(* Logix 5000 project; controller L3 vendor 1 type 14 code 92 rev 20.12; software revision 20.04 *)

TASK _11_PID2 (periodic, rate 100 ms, priority 14, watchdog 500 ms) : _11_PID2
TASK main (periodic, rate 100 ms, priority 13, watchdog 500 ms) : _2_GENERAL
TASK MainTask (continuous, watchdog 500 ms) : MainProgram
TASK pid_lent (periodic, rate 1000 ms, priority 15, watchdog 500 ms) : pid_dec

MODULES
   Local : vendor 1 type 14 code 92 (ICP 0, rev 20.12)
       : 1756-IB16 (ICP 1, rev 3.1, Input RPI 20 ms)
           Local:1:I.DATA.8   // pmp run
       : 1756-OB32 (ICP 3, rev 3.1, Output RPI 20 ms)
           Local:3:O.DATA.0   // START/STOP DRIVE POMP WKK
           Local:3:O.DATA.1   // VRIJGAVE POMP WKK
       : 1756-IF8 (ICP 2, rev 1.1, Input RPI 200 ms)
       : 1756-OF4 (ICP 4, rev 1.1, Output RPI 100 ms)
      L3_usine : 1756-EN2T (ICP 6, Ethernet 192.168.3.161, rev 2.1)
         STAT_usine : 1756-ENBT (Ethernet 192.168.3.162, rev 6.1)
            STAT : 1756-L72 (ICP 0, rev 20.1, $879c264d$ RPI 250 ms)
         EtherNet_Bridge : 1756-ENBT (Ethernet 192.168.3.150, rev 4.3, Output RPI 10 ms)
            WKK : vendor 1 type 14 code 92 (ICP 2, rev 20.12, $f706532b$ RPI 250 ms)
      IO : 1756-EN2T (ICP 5, Ethernet 192.168.1.2, rev 2.1)
         IO_decap : 1794-AENTR (Ethernet 192.168.1.6, rev 1.1, Output RPI 20 ms)
            decap_DO_3 : vendor 1 type 7 code 35 (Flex 3, rev 1.1)
            decap_DI_2 : 1794-IB16 (Flex 2, rev 1.1)
            decap_AI_0 : vendor 1 type 10 code 30 (Flex 0, rev 1.1, Input RPI 80 ms)
            decap_AO_1 : vendor 1 type 10 code 31 (Flex 1, rev 1.1, Output RPI 80 ms)
         R2 : vendor 1 type 12 code 228 (Ethernet 192.168.1.4, rev 1.1)
             : vendor 1 type 117 code 6 (SLCChassis 10, rev 1.1, StandardDataDriven RPI 20 ms)
             : vendor 1 type 117 code 6 (SLCChassis 9, rev 1.1, StandardDataDriven RPI 20 ms)
             : vendor 1 type 116 code 24 (SLCChassis 2, rev 1.1, StandardDataDriven RPI 20 ms)
                 R2:2:O.DATA.0   // CONSIGNE SORTIE -5% pg78
                 R2:2:O.DATA.1   // CONSIGNE SORTIE +5% pg78
                 R2:2:O.DATA.2   // CONSIGNE SORTIE -20% pg78
                 R2:2:O.DATA.3   // CONSIGNE SORTIE +20% pg78
                 R2:2:O.DATA.4   // CONSIGNE SORTIE 0 pg78
                 R2:2:O.DATA.5   // LP8 POTENTIOMETRE ENR POSITION incorrecte pg80
                 R2:2:O.DATA.6   // POTENTIOMETRE ENROULEUSE MIN pg80
                 R2:2:O.DATA.7   // LP6 TRS ACCU EXTREME VIDE pg82
                 R2:2:O.DATA.8   // TRS pg83
                 R2:2:O.DATA.9   // JOG -> BS4 pg85
                 R2:2:O.DATA.10   // JOG <- BS4 pg85
                 R2:2:O.DATA.11   // VERROUILAGE CISAILLE SORTIE pg87
                 R2:2:O.DATA.12   // REGLAGE TRACTION pg 93
                 R2:2:O.DATA.13   // QUEUE DE BANDE ENROULEUSE pg94
                 R2:2:O.DATA.14   // JOG -> ENR pg94.1
                 R2:2:O.DATA.15   // JOG <- ENR pg94.1
                 R2:2:O.POINT_0   // n,bvch
             : vendor 1 type 116 code 24 (SLCChassis 6, rev 1.1, StandardDataDriven RPI 20 ms)
                 R2:6:O.DATA.0   // lampe verte
                 R2:6:O.DATA.1   // bell
                 R2:6:O.DATA.2   // lampe orange
                 R2:6:O.DATA.3   // lampe rouge
                 R2:6:O.DATA.4   // lampe bleu
                 R2:6:O.DATA.5   // vann apport soude décapage
                 R2:6:O.DATA.6   // res
                 R2:6:O.DATA.7   // res
                 R2:6:O.DATA.8   // res
                 R2:6:O.DATA.9   // res
                 R2:6:O.DATA.10   // res
                 R2:6:O.DATA.11   // res
                 R2:6:O.DATA.12   // res
                 R2:6:O.DATA.13   // res
                 R2:6:O.DATA.14   // res
                 R2:6:O.DATA.15   // reserve pour vanne acide
                 R2:6:O.POINT_0   // lampe verte
                 R2:6:O.POINT_1   // bell
                 R2:6:O.POINT_2   // lampe orange
                 R2:6:O.POINT_3   // lampe rouge
                 R2:6:O.POINT_4   // lampe bleu
                 R2:6:O.POINT_5   // vann apport soude décapage
                 R2:6:O.POINT_15   // reserve pour vanne acide
             : vendor 1 type 116 code 3 (SLCChassis 7, rev 1.1, StandardDataDriven RPI 20 ms)
                 R2:7:I.DATA.0   // vanne apport soude ouverte
                 R2:7:I.DATA.1   // vanne apport soude fermée
                 R2:7:I.DATA.2   // t° redresseur T1 R2
                 R2:7:I.DATA.3   // t° redresseur T2 R2
                 R2:7:I.DATA.4   // t° redresseur T1 R3
                 R2:7:I.DATA.5   // t° redresseur T2 R3
                 R2:7:I.DATA.6   // t° redresseur T1 R4
                 R2:7:I.DATA.7   // t° redresseur T2 R4
                 R2:7:I.DATA.8   // t° redresseur T1 R1
                 R2:7:I.DATA.9   // t° redresseur T2 R1
                 R2:7:I.POINT_0   // vanne apport soude ouverte
                 R2:7:I.POINT_1   // vanne apport soude fermée
                 R2:7:I.POINT_2   // t° redresseur T1 R2
                 R2:7:I.POINT_3   // t° redresseur T2 R2
                 R2:7:I.POINT_4   // t° redresseur T1 R3
                 R2:7:I.POINT_5   // t° redresseur T2 R3
                 R2:7:I.POINT_6   // t° redresseur T1 R4
                 R2:7:I.POINT_7   // t° redresseur T2 R4
                 R2:7:I.POINT_8   // t° redresseur T1 R1
                 R2:7:I.POINT_9   // t° redresseur T2 R1
             : vendor 1 type 116 code 3 (SLCChassis 1, rev 1.1, StandardDataDriven RPI 20 ms)
                 R2:1:I.DATA.0   // TRE ACCU EXTREMEVIDE
                 R2:1:I.DATA.1   // TRE en SERVICE
                 R2:1:I.DATA.2   // TRE MAN/COORD.
                 R2:1:I.DATA.3   // AUTORISATION JOG BS2
                 R2:1:I.DATA.4   // AUTORISATION JOG BS3
                 R2:1:I.DATA.5   // MARCHE SORTIE
                 R2:1:I.DATA.6   // MARCHE SORTIE
                 R2:1:I.DATA.7   // ARRET SORTIE
                 R2:1:I.DATA.8   // SORTIE COORD.
                 R2:1:I.DATA.9   // SORTIE MANU
                 R2:1:I.DATA.10   // REPRISE MANU SORTIE
                 R2:1:I.DATA.11   // ENR POTENT.POSITION MAX
                 R2:1:I.DATA.12   // ENR POTENT.POSITION MIN
                 R2:1:I.DATA.13   // TRS RALENTSSEMENT
                 R2:1:I.DATA.14   // TRS POSITION TRAVAIL ARRIERE
                 R2:1:I.DATA.15   // TRS POSITION TRAVAIL AVANT
                 R2:1:I.POINT_0   // tdwsrdrw
             : vendor 1 type 117 code 6 (SLCChassis 8, rev 1.1, StandardDataDriven RPI 20 ms)
             : vendor 1 type 116 code 3 (SLCChassis 3, rev 1.1, StandardDataDriven RPI 20 ms)
                 R2:3:I.DATA.0   // TRS ACCU VIDE
                 R2:3:I.DATA.1   // TRS ACCU REMPLI
                 R2:3:I.DATA.2   // TRS ACCU REMPLI EXTREME
                 R2:3:I.DATA.3   // TRS ACCU VIDE EXTREME
                 R2:3:I.DATA.4   // TRS en service
                 R2:3:I.DATA.5   // TRS
                 R2:3:I.DATA.6   // JOG -> BS4
                 R2:3:I.DATA.7   // JOG <- BS4
                 R2:3:I.DATA.8   // BS4M N=0
                 R2:3:I.DATA.9   // BS3M N=0
                 R2:3:I.DATA.10   // QUEUE DE BANDE ENROULEUSE ON
                 R2:3:I.DATA.11   // QUEUE DE BANDE ENROULEUSE OFF
                 R2:3:I.DATA.12   // JOG -> ENR
                 R2:3:I.DATA.13   // JOG <- ENR
                 R2:3:I.DATA.14   // BP POSITIONNER ENR
                 R2:3:I.DATA.15   // ENROULEUSE POSITIONNEE
             : vendor 1 type 117 code 11 (SLCChassis 11, rev 1.1, StandardDataDriven RPI 20 ms)
             : vendor 1 type 116 code 3 (SLCChassis 5, rev 1.1, StandardDataDriven RPI 20 ms)
                 R2:5:I.DATA.0   // N=0 ENR
                 R2:5:I.DATA.1   // RAZ DIAMETRE ENROULEUSE
                 R2:5:I.DATA.2   // MANDRIN EXPANSE
                 R2:5:I.DATA.3   // ready drive ventilateur 03
                 R2:5:I.DATA.4   // ready drive ventilateur 2
                 R2:5:I.DATA.5   // ready drive ventilateur 01
                 R2:5:I.DATA.6   // protection drive ventilateur 03
                 R2:5:I.DATA.7   // protection drive ventilateur 2
                 R2:5:I.DATA.8   // protection drive ventilateur 01
                 R2:5:I.POINT_0   // N=0 ENR
                 R2:5:I.POINT_1   // RAZ DIAMETRE ENROULEUSE
                 R2:5:I.POINT_2   // MANDRIN EXPANSE
                 R2:5:I.POINT_3   // ready drive ventilateur 03
                 R2:5:I.POINT_4   // ready drive ventilateur 2
                 R2:5:I.POINT_5   // ready drive ventilateur 01
                 R2:5:I.POINT_6   // protection drive ventilateur 03
                 R2:5:I.POINT_7   // protection drive ventilateur 2
                 R2:5:I.POINT_8   // protection drive ventilateur 01
             : vendor 1 type 116 code 24 (SLCChassis 4, rev 1.1, StandardDataDriven RPI 20 ms)
                 R2:4:O.DATA.0   // POSITIONNER MANDRIN ENR pg94.1
                 R2:4:O.DATA.1   // RAZ DIAMETRE ENR pg96
                 R2:4:O.DATA.2   // klaxon demarrage ligne
                 R2:4:O.DATA.3   // M/A VENTILATEUR 03
                 R2:4:O.DATA.4   // M/A VENTILATEUR 2
                 R2:4:O.DATA.5   // M/A VENTILATEUR 01
                 R2:4:O.DATA.6   // VANNE VIDANGE TOURS
                 R2:4:O.DATA.7   // M/A PMP DOSEUSE TOUR REFROIDISSEMENT
                 R2:4:O.POINT_0   // POSITIONNER MANDRIN ENR pg94.1
                 R2:4:O.POINT_1   // RAZ DIAMETRE ENR pg96
                 R2:4:O.POINT_2   // klaxon demarrage ligne
                 R2:4:O.POINT_3   // M/A VENTILATEUR 03
                 R2:4:O.POINT_4   // M/A VENTILATEUR 2
                 R2:4:O.POINT_5   // M/A VENTILATEUR 01
                 R2:4:O.POINT_6   // VANNE VIDANGE TOURS
                 R2:4:O.POINT_7   // M/A PMP DOSEUSE TOUR REFROIDISSEMENT
         R1 : vendor 1 type 12 code 228 (Ethernet 192.168.1.3, rev 1.1)
             : vendor 1 type 116 code 3 (SLCChassis 6, rev 1.1, StandardDataDriven RPI 20 ms)
                 R1:6:I.DATA.0   // DEFAUT CONVERTISSEUR
                 R1:6:I.DATA.1   // ACQUIT KLAXON
                 R1:6:I.DATA.2   // TENSION 24 V PAS OK
                 R1:6:I.DATA.3   // N>N0
                 R1:6:I.DATA.4   // RUPTURE BANDE ENTREE
                 R1:6:I.DATA.5   // RUPTURE BANDE SORTIE
                 R1:6:I.DATA.6   // FREIN DEROULEUSE 1
                 R1:6:I.DATA.7   // FREIN DEROULEUSE 2
                 R1:6:I.DATA.8   // JOG <- BS1 + DEC
                 R1:6:I.DATA.9   // JOG -> BS1 + DEC
                 R1:6:I.DATA.10   // JOG <- DEC
                 R1:6:I.DATA.11   // JOG -> DEC
                 R1:6:I.DATA.12   // DEC N<N0
                 R1:6:I.DATA.13   // BS1M N<N0
                 R1:6:I.DATA.14   // BS2M N<N0
                 R1:6:I.DATA.15   // CISAILLE ENTREE BASSE
                 R1:6:I.POINT_0   // dsgt erqe
             : vendor 1 type 116 code 24 (SLCChassis 7, rev 1.1, StandardDataDriven RPI 20 ms)
                 R1:7:O.DATA.0   // RUN TEMPO pg38
                 R1:7:O.DATA.1   // FERMER PINCEUR pg39
                 R1:7:O.DATA.2   // LP6 RUPTURE BANDE pg39
                 R1:7:O.DATA.3   // JOG -> DEC pg55
                 R1:7:O.DATA.4   // JOG <- DEC pg55
                 R1:7:O.DATA.5   // N<N0 DEC pg57
                 R1:7:O.DATA.6   // LP4 M/A ENTREE pg60
                 R1:7:O.DATA.7   // LP4 ENTREE COORDONNEE pg61
                 R1:7:O.DATA.8   // LP4 ENTREE MANUEL pg61
                 R1:7:O.DATA.9   // MAN/COORD. ENTREE pg62
                 R1:7:O.DATA.10   // CONSIGNE ENTREE-5% pg63
                 R1:7:O.DATA.11   // CONSIGNE ENTREE+5% pg63
                 R1:7:O.DATA.12   // CONSIGNE ENTREE-20% pg63
                 R1:7:O.DATA.13   // CONSIGNE ENTREE+20% pg63
                 R1:7:O.DATA.14   // CONSIGNE ENTREE pg63
                 R1:7:O.DATA.15   // JOG <- BS1 pg66
                 R1:7:O.POINT_0   // vgcf
             : vendor 1 type 116 code 3 (SLCChassis 3, rev 1.1, StandardDataDriven RPI 20 ms)
                 R1:3:I.DATA_0   // EMG 2
                 R1:3:I.DATA_1   // EMG 3
                 R1:3:I.DATA_10   // TRE PRET REFERENCE
                 R1:3:I.DATA_11   // BS2M PRET REFERENCE
                 R1:3:I.DATA_12   // BS3M PRET REFERENCE
                 R1:3:I.DATA_13   // TRS PRET REFERENCE
                 R1:3:I.DATA_14   // BS4M PRET REFERENCE
                 R1:3:I.DATA_15   // ENR PRET REFERENCE
                 R1:3:I.DATA_2   // bp marche ligne
                 R1:3:I.DATA_3   // BP STOP
                 R1:3:I.DATA_4   // DEC ENCLENCHE
                 R1:3:I.DATA_5   // LIGNE ENCLENCHEE
                 R1:3:I.DATA_6   // READY FOR RUN
                 R1:3:I.DATA_7   // BP RUN
                 R1:3:I.DATA_8   // AEC PRET REFERENCE
                 R1:3:I.DATA_9   // BS1M PRET REFERENCE
                 R1:3:I.POINT_0   // dxfh
             : vendor 1 type 116 code 3 (SLCChassis 1, rev 1.1, StandardDataDriven RPI 20 ms)
                 R1:1:I.DATA.0   // bp start groupe hydraulique entrée
                 R1:1:I.DATA.1   // bp stop groupe hydraulique entrée
                 R1:1:I.DATA.2   // pression groupe hydraulique entrée 100 bars
                 R1:1:I.DATA.3   // pression groupe hydraulique entrée 70 bars
                 R1:1:I.DATA.4   // niveau groupe hydraulique entrée
                 R1:1:I.DATA.5   // by pass groupe hydraulique entrée
                 R1:1:I.DATA.6   // by pass groupe hydraulique sortie
                 R1:1:I.DATA.7   // bp start groupe hydraulique sortie
                 R1:1:I.DATA.8   // bp stop groupe hydraulique sortie
                 R1:1:I.DATA.9   // 100 BARS GROUPE HYDR.SORTIE
                 R1:1:I.DATA.10   // pression groupe hydraulique sortie 70 bars
                 R1:1:I.DATA.11   // niveau groupe hydraulique sortie
                 R1:1:I.DATA.12   // réarmement signalisation
                 R1:1:I.DATA.13   // pressostat air comprimé
                 R1:1:I.DATA.14   // centrage ok
                 R1:1:I.DATA.15   // centrage EMG 1
                 R1:1:I.POINT_0   // bp start groupe hydraulique entrée
                 R1:1:I.POINT_1   // bp stop groupe hydraulique entrée
                 R1:1:I.POINT_2   // pression groupe hydraulique entrée 100 bars
                 R1:1:I.POINT_3   // pression groupe hydraulique entrée 70 bars
                 R1:1:I.POINT_4   // niveau groupe hydraulique entrée
                 R1:1:I.POINT_6   // by pass groupe hydraulique sortie
                 R1:1:I.POINT_5   // by pass groupe hydraulique entrée
                 R1:1:I.POINT_7   // bp start groupe hydraulique sortie
                 R1:1:I.POINT_8   // bp stop groupe hydraulique sortie
                 R1:1:I.POINT_9   // 100 BARS GROUPE HYDR.SORTIE
                 R1:1:I.POINT_10   // pression groupe hydraulique sortie 70 bars
                 R1:1:I.POINT_11   // niveau groupe hydraulique sortie
                 R1:1:I.POINT_12   // réarmement signalisation
                 R1:1:I.POINT_13   // pressostat air comprimé
                 R1:1:I.POINT_14   // centrage ok
                 R1:1:I.POINT_15   // centrage EMG 1
             : vendor 1 type 116 code 24 (SLCChassis 9, rev 1.1, StandardDataDriven RPI 20 ms)
                 R1:9:O.DATA.0   // JOG -> BS1 pg66
                 R1:9:O.DATA.1   // LP4 TRE RALENTISSEMENT pg68
                 R1:9:O.DATA.2   // LP6 TRE ACCU VIDE pg69
                 R1:9:O.DATA.3   // TRE MAN/COORDON. pg70
                 R1:9:O.DATA.4   // AUTORISATION JOG BS2 pg 72
                 R1:9:O.DATA.5   // AUTORISATION JOG BS3 pg70
                 R1:9:O.DATA.6   // LP8 MARCHE SORTIE pg74
                 R1:9:O.DATA.7   // LP7 MARCHE SORTIE pg74
                 R1:9:O.DATA.8   // LP7 SORTIE MANU pg75
                 R1:9:O.DATA.9   // LP7 SORTIE COORD. pg75
                 R1:9:O.DATA.10   // LP8 NOUVELLE BOBINE SORTIE pg75
                 R1:9:O.DATA.11   // ENR DEBUT FIN DE BOBINE pg76
                 R1:9:O.DATA.12   // CONS. SORTIE MAN/COORD. pg77
                 R1:9:O.DATA.13   // CONSIGNE SORTIE MANU pg77
                 R1:9:O.DATA.14   // CONSIGNE SORTIE MARCHE MANU pg77
                 R1:9:O.DATA.15   // CONSIGNE SORTIE pg77
                 R1:9:O.POINT_0   // hfgfh
             : vendor 1 type 116 code 24 (SLCChassis 4, rev 1.1, StandardDataDriven RPI 20 ms)
                 R1:4:O.DATA.0   // DRIVE ON pg16.1
                 R1:4:O.DATA.1   // ARRET pg17
                 R1:4:O.DATA.2   // AUXILIAIRE 1 ARRET pg17
                 R1:4:O.DATA.3   // AUXILIAIRE 2 ARRET pg17
                 R1:4:O.DATA.4   // LP6 DRIVE ENCLENCHE pg18
                 R1:4:O.DATA.5   // LP6 READY FOR RUN pg18.1
                 R1:4:O.DATA.6   // RUN pg20
                 R1:4:O.DATA.7   // MARCHE SYNCHRO DEC pg21
                 R1:4:O.DATA.8   // MARCHE SYNCHRO BS1 pg21
                 R1:4:O.DATA.9   // MARCHE SYNCHRO TRE pg21
                 R1:4:O.DATA.10   // MARCHE SYNCHRO BS2 pg21
                 R1:4:O.DATA.11   // MARCHE SYNCHRO BS3 pg21
                 R1:4:O.DATA.12   // MARCHE SYNCHRO TRS pg21
                 R1:4:O.DATA.13   // MARCHE SYNCHRO BS4 pg21
                 R1:4:O.DATA.14   // MARCHE SYNCHRO ENR pg21
                 R1:4:O.DATA.15   // LP6 MARCHE COORDONNEE pg22
                 R1:4:O.POINT_0   // n cb
             : vendor 1 type 116 code 3 (SLCChassis 8, rev 1.1, StandardDataDriven RPI 20 ms)
                 R1:8:I.DATA.0   // TABLE CISAILLE ENTREE OK
                 R1:8:I.DATA.1   // BP MARCHE ENTREE
                 R1:8:I.DATA.2   // BP MARCHE ENTREE
                 R1:8:I.DATA.3   // BP ARRET ENTREE
                 R1:8:I.DATA.4   // BP ENTREE COORDONNE
                 R1:8:I.DATA.5   // BP ENTREE MANU
                 R1:8:I.DATA.6   // POTENTIOMETRE ENTREE POSITION MAX
                 R1:8:I.DATA.7   // POTENTIOMETRE ENTREE POSITION MIN
                 R1:8:I.DATA.8   // JOG <-BS1
                 R1:8:I.DATA.9   // JOG ->BS1
                 R1:8:I.DATA.10   // TRE RALENTISSEMENT
                 R1:8:I.DATA.11   // TRE POSITION TRAVAIL AVANT
                 R1:8:I.DATA.12   // TRE POSITION TRAVAIL ARRIERE
                 R1:8:I.DATA.13   // TRE ACCU REMPLI
                 R1:8:I.DATA.14   // TRE ACCU VIDE
                 R1:8:I.DATA.15   // TRE ACCU EXTREME REMPLI
                 R1:8:I.POINT_0   // ;,vn
            O2 : vendor 1 type 116 code 24 (SLCChassis 2, rev 1.1, StandardDataDriven RPI 20 ms)
                 R1:2:O.DATA.0   // n<n0 pg37
                 R1:2:O.DATA.1   // LP6 marche groupe hydraulique entrée pg8
                 R1:2:O.DATA.2   // marche groupe hydraulique entrée pg11
                 R1:2:O.DATA.3   // autorisation alimentation tension de groupe Hydraulique entrée
                 R1:2:O.DATA.4   // vanne mise en pression groupe hydraumique entrée pg8
                 R1:2:O.DATA.5   // LP6 marche groupe hydraulique sortie pg9
                 R1:2:O.DATA.6   // marche groupe hydraulique sortie pg11
                 R1:2:O.DATA.7   // autorisation alimentation tension de groupe Hydraulique sortie
                 R1:2:O.DATA.8   // vanne mise en pression groupe hydraumique sortie pg9
                 R1:2:O.DATA.9   // LP6 defaut pression groupe hydraulique entrée pg10
                 R1:2:O.DATA.10   // LP6 défaut niveau groupe hydraulique entrée pg10
                 R1:2:O.DATA.11   // LP6 défaut pression groupe hydraulique sortie 70 bars
                 R1:2:O.DATA.12   // LP6 défaut niveau groupe hydraulique entrée pg10
                 R1:2:O.DATA.13   // LP6 défaut pression air comprimé pg11.1
                 R1:2:O.DATA.14   // drive on pg16
                 R1:2:O.DATA.15   // LP6 demande drive on
                 R1:2:O.POINT_0   // n<n0 pg37
                 R1:2:O.POINT_1   // LP6 marche groupe hydraulique entrée pg8
                 R1:2:O.POINT_2   // marche groupe hydraulique entrée pg11
                 R1:2:O.POINT_3   // autorisation alimentation tension de groupe Hydraulique entrée
                 R1:2:O.POINT_4   // vanne mise en pression groupe hydraumique entrée pg8
                 R1:2:O.POINT_5   // LP6 marche groupe hydraulique sortie pg9
                 R1:2:O.POINT_6   // marche groupe hydraulique sortie pg11
                 R1:2:O.POINT_7   // autorisation alimentation tension de groupe Hydraulique sortie
                 R1:2:O.POINT_8   // vanne mise en pression groupe hydraumique sortie pg9
                 R1:2:O.POINT_9   // LP6 defaut pression groupe hydraulique entrée pg10
                 R1:2:O.POINT_10   // LP6 défaut niveau groupe hydraulique entrée pg10
                 R1:2:O.POINT_12   // LP6 défaut niveau groupe hydraulique entrée pg10
                 R1:2:O.POINT_11   // LP6 défaut pression groupe hydraulique sortie 70 bars
                 R1:2:O.POINT_14   // drive on pg16
                 R1:2:O.POINT_13   // LP6 défaut pression air comprimé pg11.1
                 R1:2:O.POINT_15   // LP6 demande drive on
             : vendor 1 type 116 code 24 (SLCChassis 5, rev 1.1, StandardDataDriven RPI 20 ms)
                 R1:5:O.DATA.0   // LP6 PRET REFERENCE DEC pg25
                 R1:5:O.DATA.1   // LP6 PRET REFERENCE BS1 pg25
                 R1:5:O.DATA.2   // LP6 PRET REFERENCE TRE pg25
                 R1:5:O.DATA.3   // LP6 PRET REFERENCE BS2 pg25
                 R1:5:O.DATA.4   // LP6 PRET REFERENCE BS3 pg25
                 R1:5:O.DATA.5   // LP6 PRET REFERENCE TRS pg25
                 R1:5:O.DATA.6   // LP6 PRET REFERENCE BS4 pg25
                 R1:5:O.DATA.7   // LP6 PRET REFERENCE ENR pg25
                 R1:5:O.DATA.8   // LP6 PRET REFERENCE LIGNE pg25
                 R1:5:O.DATA.9   // LIGNE PRET REFERENCE pg26
                 R1:5:O.DATA.10   // LP6 DEFAUT PRET REFERENCE pg27
                 R1:5:O.DATA.11   // LP6 DEFAUT PRET REFERENCE BS2 BS3 pg27
                 R1:5:O.DATA.12   // LP6 DEFAUT MISE EN VITESSE pg27
                 R1:5:O.DATA.13   // LP6 DEFAUT CONVERTISSEUR pg28
                 R1:5:O.DATA.14   // KLAXON pg30
                 R1:5:O.DATA.15   // LP6 ALIM. 24 V OK pg33
                 R1:5:O.POINT_0   // ;: ,hwfd
         R3 : vendor 1 type 12 code 228 (Ethernet 192.168.1.5, rev 1.1)
             : vendor 1 type 116 code 6 (SLCChassis 7, rev 1.1, StandardDataDriven RPI 20 ms)
                 R3:7:I.POINT_0   // v cxbvwc
             : vendor 1 type 117 code 11 (SLCChassis 2, rev 1.1, StandardDataDriven RPI 20 ms)
                 R3:2:O.CHANNEL_0_OUTPUT   // wxvc<
             : vendor 1 type 117 code 6 (SLCChassis 6, rev 1.1, StandardDataDriven RPI 20 ms)
                 R3:6:I.CHANNEL_0_DATA   // vwx
             : vendor 1 type 117 code 6 (SLCChassis 3, rev 1.1, StandardDataDriven RPI 20 ms)
                 R3:3:I.CHANNEL_0_DATA   // vwxc
             : vendor 1 type 116 code 6 (SLCChassis 4, rev 1.1, StandardDataDriven RPI 20 ms)
                 R3:4:I.DATA.0   // vanne chauffe degrai open
                 R3:4:I.DATA.1   // vanne chauffe degrai closed
                 R3:4:I.DATA.2   // vanne chauffe decapa open
                 R3:4:I.DATA.3   // vanne chauffe decapa close
                 R3:4:I.DATA.4   // vanne froid decapage open
                 R3:4:I.DATA.5   // vanne froid decapage closed
                 R3:4:I.DATA.6   // fc open vanne ano
                 R3:4:I.DATA.7   // fc closed vanne ano
                 R3:4:I.DATA.8   // vanne chauffage colm open
                 R3:4:I.DATA.9   // vanne chauffage colm closed
                 R3:4:I.DATA.10   // vanne 2 chauffage co open
                 R3:4:I.DATA.11   // vanne 2 chauffage co closed
                 R3:4:I.DATA.12   // P1 T37 DECAPAGE RUN
                 R3:4:I.DATA.13   // P1 T37 DECAPAGE PROTECTION
                 R3:4:I.DATA.14   // P2 DECAPAGE RUN
                 R3:4:I.DATA.15   // P2 DECAPAGE PROTECTION
                 R3:4:I.DATA.16   // Naoh L3VA1 FC O
                 R3:4:I.DATA.17   // Naoh L3VA1 FC f
                 R3:4:I.DATA.18   // Naoh L3VA2 FC O
                 R3:4:I.DATA.19   // Naoh L3VA2 FC F
                 R3:4:I.DATA.20   // Naoh L3VA3 FC O
                 R3:4:I.DATA.21   // Naoh L3VA3 FC F
                 R3:4:I.DATA.22   // Naoh L3VA4 FC O
                 R3:4:I.DATA.23   // Naoh L3VA4 FC F
                 R3:4:I.DATA.24   // re
                 R3:4:I.DATA.25   // re
                 R3:4:I.DATA.26   // NaOH FLOW METER PULSE 0.1 M³
                 R3:4:I.DATA.27   // laveur fumée ok
                 R3:4:I.DATA.28   // fc vanne apport acide ano open
                 R3:4:I.DATA.29   // fc vanne apport acide ano close
                 R3:4:I.DATA.30   // fc vanne apport acide neutral open
                 R3:4:I.DATA.31   // fc vanne apport acide neutral close
                 R3:4:I.POINT_0   // vanne chauffe degrai open
                 R3:4:I.POINT_1   // vanne chauffe degrai closed
                 R3:4:I.POINT_2   // vanne chauffe decapa open
                 R3:4:I.POINT_3   // vanne chauffe decapa close
                 R3:4:I.POINT_4   // vanne froid decapage open
                 R3:4:I.POINT_5   // vanne froid decapage closed
                 R3:4:I.POINT_6   // fc open vanne ano
                 R3:4:I.POINT_7   // fc closed vanne ano
                 R3:4:I.POINT_8   // vanne chauffage colm open
                 R3:4:I.POINT_9   // vanne chauffage colm closed
                 R3:4:I.POINT_10   // vanne 2 chauffage co open
                 R3:4:I.POINT_11   // vanne 2 chauffage co closed
                 R3:4:I.POINT_12   // P1 T37 DECAPAGE RUN
                 R3:4:I.POINT_13   // P1 T37 DECAPAGE PROTECTION
                 R3:4:I.POINT_14   // P2 DECAPAGE RUN
                 R3:4:I.POINT_15   // P2 DECAPAGE PROTECTION
                 R3:4:I.POINT_16   // Naoh L3VA1 FC O
                 R3:4:I.POINT_17   // Naoh L3VA1 FC f
                 R3:4:I.POINT_18   // Naoh L3VA2 FC O
                 R3:4:I.POINT_19   // Naoh L3VA2 FC F
                 R3:4:I.POINT_20   // Naoh L3VA3 FC O
                 R3:4:I.POINT_21   // Naoh L3VA3 FC F
                 R3:4:I.POINT_22   // Naoh L3VA4 FC O
                 R3:4:I.POINT_23   // Naoh L3VA4 FC F
                 R3:4:I.POINT_26   // NaOH FLOW METER PULSE 0.1 M³
                 R3:4:I.POINT_27   // laveur fumée ok
                 R3:4:I.POINT_24   // fc vanne apport acide ano open
                 R3:4:I.POINT_28   // fc vanne apport acide ano open
                 R3:4:I.POINT_29   // fc vanne apport acide ano close
                 R3:4:I.POINT_30   // fc vanne apport acide neutral open
                 R3:4:I.POINT_31   // fc vanne apport acide neutral close
             : vendor 1 type 117 code 11 (SLCChassis 1, rev 1.1, StandardDataDriven RPI 20 ms)
                 R3:1:O.CHANNEL_0_OUTPUT   // SORTIE VANNE DEGRAISSAGE
                 R3:1:O.CHANNEL_1_OUTPUT   // max etait 31850
                 R3:1:O.CHANNEL_2_OUTPUT   // 6500 le 21/2/16
             : vendor 1 type 116 code 30 (SLCChassis 5, rev 1.1, StandardDataDriven RPI 20 ms)
                 R3:5:O.POINT_1   // va2
                 R3:5:O.POINT_2   // va3
                 R3:5:O.DATA.0   // va1
                 R3:5:O.DATA.1   // va2
                 R3:5:O.DATA.2   // va3
                 R3:5:O.DATA.3   // va4
                 R3:5:O.DATA.4   // vanne apport acide ano
                 R3:5:O.DATA.5   // apport level colmatage
                 R3:5:O.DATA.6   // vanne apport acide neutral
                 R3:5:O.DATA.7   // res
                 R3:5:O.DATA.8   // autoristion pompage colmatage
                 R3:5:O.DATA.9   // res
                 R3:5:O.DATA.10   // res
                 R3:5:O.DATA.11   // res
                 R3:5:O.DATA.12   // res
                 R3:5:O.DATA.13   // se ferme diminue chauffage
                 R3:5:O.DATA.14   // pour augmenter le chauffage
                 R3:5:O.DATA.15   // res
                 R3:5:O.DATA.16   // res
                 R3:5:O.DATA.17   // res
                 R3:5:O.DATA.18   // res
                 R3:5:O.DATA.19   // res
                 R3:5:O.DATA.20   // res
                 R3:5:O.DATA.21   // res
                 R3:5:O.DATA.22   // res
                 R3:5:O.DATA.23   // res
                 R3:5:O.DATA.24   // res
                 R3:5:O.DATA.25   // res
                 R3:5:O.DATA.26   // res
                 R3:5:O.DATA.27   // res
                 R3:5:O.DATA.28   // res
                 R3:5:O.DATA.29   // res
                 R3:5:O.DATA.30   // res
                 R3:5:O.DATA.31   // res
                 R3:5:O.POINT_0   // va1
                 R3:5:O.POINT_16   // vanne refroidir decapage ouvrir
                 R3:5:O.POINT_17   // vanne refroidir decapage fermer
                 R3:5:O.POINT_3   // va4
                 R3:5:O.POINT_4   // vanne apport acide ano
                 R3:5:O.POINT_5   // pompe colmatage apport level colmatage
                 R3:5:O.POINT_6   // vanne apport acide neutral
                 R3:5:O.POINT_8   // autoristion pompage colmatage
                 R3:5:O.POINT_13   // se ferme diminue chauffage decapage
                 R3:5:O.POINT_14   // pour augmenter le chauffage decapage
END_MODULES

ADD_ON_INSTRUCTION integrat   (* revision 1.0 *)
VAR_INPUT
   rate : DINT; {required}
END_VAR
VAR_OUTPUT
   oai : DINT; {access Read Only, required}
END_VAR
VAR_INPUT
   AI : DINT; {required}
END_VAR
VAR
   memo : REAL; {access None}
   memo1 : REAL; {access None}
   rate1 : DINT; {access None}
   memo2 : REAL; {access None}
END_VAR

ROUTINE Logic   (* ladder *)
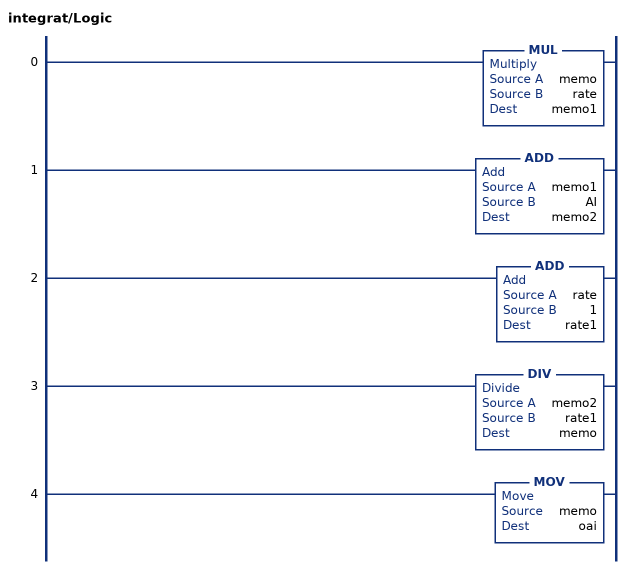
   0: MUL(memo,rate,memo1);
   1: ADD(memo1,AI,memo2);
   2: ADD(rate,1,rate1);
   3: DIV(memo2,rate1,memo);
   4: MOV(memo,oai);
END_ROUTINE
END_ADD_ON_INSTRUCTION

ADD_ON_INSTRUCTION SCP   (* revision 1.2, vendor Rockwell Automation *)
VAR_INPUT
   Input : REAL; {required}
   Input_Min : REAL; {required}
   Input_Max : REAL; {required}
   Scaled_Min : REAL; {required}
   Scaled_Max : REAL; {required}
END_VAR
VAR_OUTPUT
   Output : REAL; {access Read Only, required}
END_VAR
VAR
   Rate : REAL;
END_VAR

ROUTINE Logic   (* ladder *)
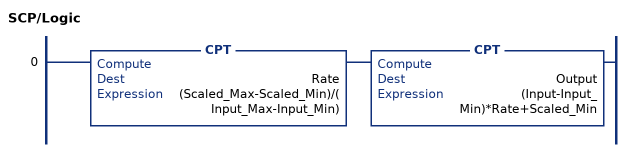
   0: CPT(Rate,(Scaled_Max-Scaled_Min)/(Input_Max-Input_Min))CPT(Output,(Input-Input_Min)*Rate+Scaled_Min);
END_ROUTINE
END_ADD_ON_INSTRUCTION

VAR_GLOBAL   (* controller tags *)
   A_CV_COLMAT : REAL := 32767.002;
   A_CV_DEC_CH : REAL := 31208.0;
   A_CV_DEG : REAL := 32200.0;
   A_LVL_DEC : REAL := 464.33203;
   A_T_DEG : REAL := 357.31726;
   anonew : BOOL;
   aux_cond_tour : REAL := 1629.6979;
   aux_dec : integrat := (rate := 2000, oai := 454, AI := 453);
   aux_dec_froid : REAL := 9558.0;
   AUX_LVL_DEC : REAL := 65.38491;
   aux_manu_dec_fr : REAL := 6500.0;
   aux_spano : DINT := 367;
   AUX_wkk5 : REAL;
   auxtempfroiddec : DINT := 450;
   averagge_rate_sec : DINT := 360;
   B3 : DINT[100] := ([1] := 2#0000_0000_0000_0000_1000_1000_0100_0000, [2] := 2#0000_0000_0000_0000_0100_0000_1010_0000, [3] := 2#0000_0000_0000_0000_0110_0000_0000_0000, [5] := 2#0000_0000_0000_0000_0000_0000_1000_1101, [7] := 2#0000_0000_0000_0000_0000_0000_0000_1011, [10] := 2#0000_0000_0000_0000_0000_0000_0000_0010);
        [0].1   // by pass groupehydraulique entrée
        [0].2   // by pass groupehydraulique sortie
        [0].3   // defaut avecdéclenchement1
        [0].4   // bit defaut avecdéclenchement 2
        [0].5   // demande run
        [0].6   // marche arret entrée
        [0].7   // sortie manu/coord.
        [0].8   // sortie marche/arret
        [0].9   // non coordonnée
        [0].10   // AEC pret ref
        [0].11   // defaut groupehydraulique
        [0].12   // auxiliaire defautaccu
        [0].13   // auxiliaire defautcentreur
        [0].14   // entréemanuel/coordoné
        [0].15   // auxiliaire positionpotentiomètre entrée
        [1].0   // position travailavant accu TRE
        [1].1   // auxiliaire accu TRErempli
        [1].2   // auxiliairepositionpotentiomètre ENR
        [1].3   // auxiliaire début finde bobine enrouleuse
        [1].4   // TRS accu vide
        [1].5   // TRS position travailavant
        [1].6   // one shot
        [1].7   // marche apres klaxon
        [1].8   // aux level high ano
        [1].9   // aux level low ano
        [1].11   // DEMANDE DE FROID
        [1].12   // demande de chauffedecapage
        [1].13   // températurecolmatage trop hautepour vider
        [1].15   // avec retour position
        [2].0   // marche ventilateur3
        [2].1   // marche ventilateur 2
        [2].2   // marche ventilateur1
        [2].3   // ons
        [2].4   // T° eau descent
        [2].5   // T° eau monte
        [3].0   // LINE RUN
        [3].1   // ARRET ENTRETIEN
        [3].2   // ON TOUTE LES MINUTE
        [3].14   // ons
        [4].1   // ONS
        [4].2   // marche acideouverture vanne
        [4].3   // apport acidedemande de marche
        [4].4   // demande stopacide
        [4].5   // demande acide
        [4].8   // ons
        [4].9   // demande soudel3
        [4].10   // ons
        [4].11   // demande stopsoude
        [4].12   // apport soudedemande de marche
        [4].13   // marche soudeouverture vanne
        [4].15   // ons
        [5].0   // ONS
        [5].1   // ONS
        [5].2   // ONS
        [5].3   // ons
        [5].4   // ONS
        [5].5   // ons
        [5].6   // ons
        [5].7   // ons
        [5].8   // ons
        [5].9   // ons
        [6].0   // ouvrir vanne T°dégraissage
        [6].1   // fermer vanne T°dégraissage
   BITMW2 : BOOL;
   C5 : COUNTER[5];
   chauffe_fort : BOOL;
   cligno : BOOL := 1;
   CONV_MSG_R_lancy : MESSAGE;
        MessageParameters(ServiceCode := 16#0fa2, LocalElement := NCOM[11], ...)
   CONV_MSG_W_lancy : MESSAGE;   // N9:70 dans n9:30
        MessageParameters(ServiceCode := 16#0faa, LocalElement := NCOM[0], ...)
   CONV_PID_N10_10 : PID := (CTL := -1610612736, EN := 1, CL := 1, SP := 500.0, KP := 125.0, KI := 4200.0, MAXS := 1000.0, DB := 2.0, MAXO := 100.0, UPD := 10.0, PV := 501.0, ERR := -1.0);   // *** Tag created for conversion to PID type required for instruction translation ***
   CONV_PID_N10_130 : PID := (CTL := -1610612736, EN := 1, CL := 1, SP := 948.0, KP := 300.0, KI := 1200.0, MAXS := 1000.0, DB := 2.0, MAXO := 100.0, UPD := 10.0, PV := 948.0);   // *** Tag created for conversion to PID type required for instruction translation ***
   CONV_PID_N10_170 : PID := (CTL := -503316480, EN := 1, CT := 1, CL := 1, CA := 1, SP := 600.0, KP := 100.0, KI := 100.0, MAXS := 1000.0, DB := 2.0, MAXO := 50.0, UPD := 10.0, PV := 600.0);   // *** Tag created for conversion to PID type required for instruction translation ***
   CONV_PID_N10_210 : PID;   // *** Tag created for conversion to PID type required for instruction translation ***
   CONV_PID_N10_50 : PID := (CTL := -1610612736, EN := 1, CL := 1, SP := 600.0, KP := 200.0, KI := 3200.0, MAXS := 1000.0, DB := 3.0, MAXO := 100.0, UPD := 10.0, PV := 600.0);   // *** Tag created for conversion to PID type required for instruction translation ***
   CONV_PID_N10_90 : PID := (CTL := -2113929216, EN := 1, CA := 1, SP := 372.0, KP := 350.0, KI := 155.0, MAXS := 1000.0, DB := 1.0, MAXO := 100.0, UPD := 10.0, PV := 371.0, ERR := -1.0);   // *** Tag created for conversion to PID type required for instruction translation ***
   csg_fermet_v_Dec_froid : DINT := 6500;
   CSG_N_VENTILO : REAL := 50.0;
   CV_ANO : REAL;
   cv_ch_dec : REAL;
   CV_PID_wkk : DINT := 100;
   cv_pmpano : DINT;
   cv_pmprenv : DINT := 1000;
   DateTime : DINT[7] := ([0] := 2017, [1] := 1, [2] := 30, [3] := 10, [4] := 18, [5] := 32, [6] := 368840);   // DINT array tag for retrieve wallclock time through GSV created during conversion
        [0]   // Year
        [1]   // Month
        [2]   // Day
        [3]   // Hour
        [4]   // Minute
        [5]   // Second
        [6]   // Microsecond
   dbpmpeau : DINT := 50;
   def_ready_pmp_decap_1 : BOOL;
   def_ready_pmp_decap_2 : BOOL;
   def_ready_pmpeau1 : BOOL;
   def_ready_pmpeau2 : BOOL;
   def_ready_ventilo_eau_1 : BOOL;
   def_ready_ventilo_eau_2 : BOOL;
   def_ready_ventilo_eau_3 : BOOL;
   delta_3min_dec : DINT;
   delta_cv_ano : DINT;
   delta_max_t_wkk : DINT := 40;
   delta_sp_dec : DINT := -3;
   dif_I_red : DINT;
   diff_t_ano : DINT := 1;
   dmd_run_pmp1_decap : BOOL := 1;
   dmd_run_pmp2_decap : BOOL := 1;
   F8 : REAL[100] := ([1] := 1646.4741, [2] := 1648.1678, [3] := 1648169.5, [4] := 1649816.0, [5] := 184.87717, [6] := 9243.586, [7] := 9428.463, [11] := 184.87183, [12] := 501.0, [13] := 999.9701, [14] := 500.0, [15] := 2026157.0, [16] := 558941440.0, [17] := 162.09256, [18] := 0.5628214, [19] := 2880.9004, [20] := 2881.0, [21] := 1648.0, [24] := 501.0, [25] := 346.0, [27] := 0.161631, [28] := 0.006103888, [30] := 1186.3143, [31] := 999.9893, [32] := 20.00025, [35] := 464.332, [36] := 23680.086, [37] := 464.3154, [38] := 210.11673, [39] := 210.20813, [42] := 9350.0, [43] := 1000.0, [44] := 1000.07635, [46] := 8141.2915, [47] := 0.4, [48] := 418.6163, [51] := 2527.774, [52] := 842.5913, [53] := 8.e-05, [55] := 25552.732, [56] := 824.2817, [57] := 17934.262, [58] := 854.01245, [59] := 43322.543, [60] := 849.4616, [61] := 132.85966, [62] := 132.84978, [63] := 1415.85, [64] := 1295.9202, [65] := 820.83875, [66] := 977.69604, [67] := 68.36041, [68] := 300.4381, [70] := 1.1116498, [71] := 1.1116527, [72] := 55.582638, [73] := 56.694286, [75] := 486.6102, [76] := 486.6824, [77] := 883.03955,
        [78] := 5298.0396);
        [1]   // aux.conduct tour
        [2]   // conduct tour
        [3]   // aux.conduct tour
        [4]   // aux.conduct tour
        [5]   // aux.T° ANDISATION
        [6]   // aux.T° ANDISATION
        [7]   // aux.T° ANDISATION
        [8]   // aux. i total redresseur
        [9]   // aux. i total redresseur
        [10]   // i total redresseur
        [11]   // T° ANDISATION
        [12]   // stock mazout
        [14]   // stock soude L1
        [15]   // somme débit depuis 1 h
        [16]   // memo somme debit en 1 h
        [17]   // temps en sec marche pmp doseuse
        [18]   // quantité d'eau passé en m3
        [19]   // total m3
        [20]   // place disponible soude
        [21]   // stock total soude
        [22]   // stock soude L2
        [23]   // niveau ano L1
        [24]   // T°DEGRAISSAGE
        [25]   // AUXILIAIRE T°DEGRAISSAGE
        [26]   // AUXILIAIRE T°DECAPAGE
        [27]   // AUXILIAIRE T°ano
        [28]   // AUXILIAIRE T°COLMATAGE
        [29]   // auxiliaire T° decapage froid
        [30]   // poisit vanne DEGRAISSAGE instantanné
        [31]   // auxiliaire POS VANNE COLM 1
        [32]   // position vanne décapage instantanné
        [33]   // auxiliaire TEMP DECAPAGE
        [34]   // TEMP COLMATAGE
        [35]   // auxiliaire level decap
        [36]   // auxiliaire level decap
        [37]   // auxiliaire level decap
        [38]   // T° colo entrée instantanne
        [39]   // aux temp colo
        [40]   // I redr.instanne
        [41]   // aux I redresseur
        [42]   // aux.T°decapage
        [43]   // aux.T°decapage
        [44]   // aux.T°decapage
        [45]   // TOTAL NaOH PASSER
        [46]   // TOTAL NaOH PASSER
        [47]   // TOTAL WATER PASSER
        [48]   // TOTAL WATER PASSER
        [49]   // aux temp colmat
        [51]   // t° colmat
        [52]   // t° colmat/3
        [53]   // rapport eau - aquatr initial 0.0001
        [55]   // aux temp in colm
        [56]   // aux temp in colmatage
        [57]   // aux temp colm out
        [58]   // aux temp colm out
        [59]   // aux temp colmatage milieu
        [60]   // aux temp colmatage milieu
        [62]   // aux position vanne refroid decapage
        [67]   // level neutral
        [68]   // level neutral
        [70]   // aux.VITESSE
        [71]   // VITESSE
        [72]   // aux.VITESSE
        [73]   // aux.VITESSE
        [75]   // debit echangeur decapage soude
        [76]   // debit echangeur soude
        [77]   // aux. level colmatage
        [78]   // aux. level colmatage
   fact_regul_pmpano : REAL := 1.8;
   FLOW_TOUR : DINT;
   ForceStatus : INT := 2;   // INT tag to retrieve Force enabled value through GSV created during conversion
   high_lim_pmpano : DINT := 700;
   I_chut : BOOL;
   I_mont : BOOL;
   I_R1 : REAL := 0.012971158;
   I_R2 : REAL := 0.012971158;
   I_R3 : REAL := 0.012971158;
   I_R4 : REAL := -0.012971158;
   inc_ano : DINT := 5;
   inc_ventilo : DINT := 150;
   int_CV_wkk : integrat := (rate := 250);
   INT_T_DEC : integrat := (rate := 1000, oai := 1000, AI := 1000);
   int_T_deg : integrat := (rate := 1000, oai := 346, AI := 342);
   khighano : DINT := 55;
   klowano : DINT := 55;
   kp_dec_ch : REAL := 7.0;
   L3_stat : DINT[20] := ([1] := 32784, [2] := 80, [5] := 464, [6] := 430, [8] := 4, [11] := 10, [13] := 16); {produced}
        [0]   // quantité soude demandee
        [1].0   // vers plc stock demande de soude L3
        [1].1   // vers plc stock demande d'arret apport soude
        [1].2   // vers plc stock fc vanne apport soude décapage open
        [1].3   // vers plc stock apport soude finit
        [1].4   // vers plc stock fc vanne apport soudefermee
        [1].15   // T°COLMATAGE <95°
        [2]   // quantité acide demandee
        [2].0   // vers plc stock demande de acide
        [2].1   // vers plc stock demande d'arret apport acide
        [2].2   // vers plc stock fc vanne apport acide open
        [2].3   // vers plc stock apport acide finit
        [2].4   // vers plc stock fc vanne apport acid fermee
        [2].5   // fc vanne apport acide neutral open
        [2].6   // fc vanne apport acide neutral close
        [3].0   // DEMANDE ACIDE
        [3].1   // DEMENDE ARRET ACIDE
   L3_wkkk : DINT[125] := ([0] := 527, [1] := 849, [2] := 851, [3] := 842, [4] := 9, [6] := 990, [8] := 12); {produced}
   limb_pmpeau : DINT := 450;
   limBBtano : DINT := 365;
   limBtano : DINT := 368;
   limh_pmpeau : DINT := 550;
   limhhtano : DINT := 375;
   limhtano : DINT := 375;
   low_lim_pmpano : DINT := 600;
   LVL_ANO : REAL := 119.935905;
   LVL_COLMAT : REAL := 883.87885;
   M_nbr_ventilo_ano : DINT := 1;
   mem1_i_tot : DINT;
   mem_cv_ano : DINT;
   mem_cv_pmpano : DINT := 585;
   mem_i_tot : DINT;
   mem_t_ano : DINT := 187;
   memtdec : REAL := 163307.0;
   MinorFaultBits : DINT;   // MinorFaultBits
   mot_test : DINT := 200;
   mw : BOOL;
   mwdec1 : BOOL;
   mwdec2 : BOOL;
   mwint : INT := 500;
   mwword : DINT := 32000;
   N10 : DINT[233] := ([0] := 346, [1] := 100, [4] := 346, [5] := 346, [10] := -24320, [12] := 500, [13] := 125, [14] := 4200, [17] := 1000, [19] := 2, [21] := 100, [23] := 10, [24] := 501, [25] := -1, [26] := 42, [27] := 6954, [28] := -7568, [29] := 2, [30] := 256, [32] := 500, [40] := 454, [44] := 453, [45] := 454, [50] := -24320, [52] := 600, [53] := 200, [54] := 3200, [57] := 1000, [59] := 3, [61] := 100, [63] := 10, [64] := 600, [66] := 63, [67] := 10356, [68] := 31697, [69] := 2, [70] := 26464, [72] := 600, [80] := 185, [90] := -24564, [92] := 372, [93] := 350, [94] := 155, [97] := 1000, [99] := 1, [101] := 100, [103] := 10, [104] := 371, [105] := -1, [106] := 17, [107] := 3311, [108] := -20351, [109] := 1, [110] := 31744, [112] := 372, [120] := 842, [121] := 100, [124] := 842, [125] := 841, [129] := -2,
        [130] := -24320, [132] := 948, [133] := 300, [134] := 1200, [137] := 1000, [139] := 2, [141] := 100, [143] := 10, [144] := 948, [146] := 28, [147] := 4542, [148] := -21224, [149] := 3, [150] := -13392, [152] := 948, [160] := 454, [161] := 139, [164] := 453, [170] := -23804, [172] := 600, [173] := 100, [174] := 100, [177] := 1000, [179] := 2, [181] := 50, [183] := 10, [184] := 600, [186] := 73, [187] := 11998, [188] := -11554, [189] := 2, [190] := 26464, [192] := 600);
        [0]   // T°(PV)degraissage
        [1]   // outputpid degraissage
        [2]   // output piddegraissage signé
        [3]   // LOW LIMIT DEADBANDT°DEGRAISSAGE
        [4]   // T°DEGRAISSAGEact
        [5]   // T°DEGRAISSAGEil y a 90 s
        [6]   // PID EN .001 sT°DEGRAISSAGE
        [7]   // NOMBRE PULSE 0.01SA AVOIRREGULDEGRAISSAGE
        [8]   // TEMPS OUVERTUREVANNE T°DEGRAISSAGE.01s
        [9]   // anticipationdegraissage
        [10]   // PID degraissage
        [10].1   // pid DEGRAISSAGE ENMANU
        [10].2   // change PV-SP toSp-PVpid degraissage
        [12]   // set pointdegraissage
        [22]   // Set point piddégraissage
        [26]   // control variablepid degraissage
        [40]   // T°(PV)decapageCHAUFFE
        [41]   // outputpid decapage
        [42]   // output piddecapage signé
        [43]   // LOW LIMIT DEADBANDT° DECAPAGE
        [44]   // T° DECAPAGE
        [45]   // T°DEcapAGEil y a 90 s
        [46]   // PID EN .001 sT°DECAPAGE
        [47]   // NBRE PULSE 0.04ST°DEcapAGE
        [49]   // anticipationdecapage
        [50]   // PID decapage
        [50].1   // pid DECAPAGEEN MANU
        [50].2   // change PV-SP toSp-PVpid decapage
        [52]   // set pointchauffedecapage
        [62]   // Set point piddecapage
        [66]   // control variablepid decapage
        [80]   // T°(PV)anodisation
        [81]   // outputpid anodisation
        [82]   // output pidanodisation signé
        [83]   // LOW LIMIT DEADBANDT° ANODISATION
        [84]   // LOW LIMIT DEADBANDT° ANODISATION
        [85]   // ADAPTATIONN TEMPO T°ANODISATION
        [86]   // PID EN .001 s T°anodisation
        [87]   // nbre pulse regul ano
        [88]   // TEMPS OUVERTUREVANNE T°anodisation.01s
        [90]   // PID anodisation
        [90].1   // pid ANODISATION ENMANU
        [90].2   // change PV-SP toSp-PVpid anodisation
        [92]   // set pointtemp anodpour PID
        [102]   // Set point pidanodisation
        [106]   // control variablepid anodisation
        [120]   // T° (PV)colmatage
        [121]   // outputpid colmatage
        [122]   // output pidcolmatage signé
        [123]   // LOW LIMIT DEADBANDT° colmatage
        [124]   // T° colmatage
        [125]   // T°colmatageil y a 90 s
        [126]   // PID EN .001 s T°colmatage
        [127]   // NBRE PULSE 0.04ST°colmatage
        [129]   // anticipationcolmatage
        [130]   // PID colmatage
        [130].1   // pid COLMATAGE ENMANU
        [130].2   // change PV-SP toSp-PVpid colmatage
        [132]   // set pointpid colmatage
        [142]   // Set point pidcolmatage
        [146]   // control variablepid colmatage
        [160]   // N9[10]
        [161]   // outputpid décapage froid
        [166]   // PID EN .001 s T°decapage froid
        [170]   // pid decapage froid
        [170].1   // pid decapafe froidENMANU
        [172]   // set point refroiddecapage
        [200]   // T°(PV)colo
        [210].1   // pid colo ENMANU
        [212]   // set pointcolo
   N20 : DINT[200] := ([10] := 40, [11] := 22, [12] := 23, [13] := 40, [14] := 30, [15] := 20, [16] := 20, [17] := 30, [18] := 25, [19] := 17, [20] := 12, [21] := 20, [22] := 40, [23] := 20, [24] := 20, [25] := 40, [26] := 40, [27] := 20, [28] := 20, [29] := 40, [100] := 3, [101] := 3, [102] := 66, [103] := 1, [104] := 1, [105] := 58);
        [5].1   // NEW DEFAULT ONTVET
        [5].2   // NEW DEFAULT REININGEN
        [5].3   // NEW DEFAULT NEUTRAL
        [5].4   // NEW DEFAULT ANODIS
        [5].5   // NEW DEFAULT KLEUR C
        [5].6   // NEW DEFAULT KLEUR E
        [5].7   // NEW DEFAULT COLMAT
        [5].8   // NEW DEFAULT OUTPUT
        [6].1   // DEFAULT ONTVET
        [6].2   // DEFAULT REININGEN
        [6].3   // DEFAULT NEUTRAL
        [6].4   // DEFAULT ANODIS
        [6].5   // DEFAULT KLEUR C
        [6].6   // DEFAULT KLEUR E
        [6].7   // DEFAULT COLMAT
        [6].8   // DEFAULT OUTPUT
        [9].1   // ack degrais
        [9].2   // ack decap
        [9].3   // ack neutral
        [9].4   // ack ano
        [9].5   // ack kleur chem
        [9].6   // ack kleur electro
        [9].7   // ack colm
        [9].8   // ack output
        [10]   // LLTEMPDEG
        [11]   // LTEMPDEG
        [12]   // HTEMPDEG
        [13]   // HHTEMPDEG
        [14]   // LLTEMPDEC
        [15]   // LTEMPDEC
        [16]   // HTEMPDEC
        [17]   // HHTEMPDEC
        [18]   // LLTEMPANO
        [19]   // LTEMPANO
        [20]   // HTEMPANO
        [21]   // HHTEMPANO
        [26]   // LLTEMPCOLM
        [27]   // LTEMPCOLM
        [28]   // HTEMPCOLM
        [29]   // HHTEMPCOLM
        [35].0   // temperature sensor default
        [35].1   // DEFAULT LOW LOW temperature
        [35].2   // DEFAULT LOW temperature
        [35].3   // DEFAULT HIGHT temperature
        [35].4   // DEFAULT HIGHT HIGHT temperature
        [35].5   // DEFAUT FERMETURE SERVOVANNE
        [35].6   // DEFAUT OUVERTURE SERVOVANNE
        [35].7   // protection alimentation servovanne froid degraissage
        [38].0   // PMP 1 DECAP ELETRICAL FAULT
        [38].1   // PMP 2 DECAP ELETRICAL FAULT
        [38].2   // DECAPAGE VA 1 valve position default
        [38].3   // VA2 POSITION DEFAULT
        [38].4   // Fresh NaOH valve position default
        [38].5   // LEVEL TOO HIGH main Tank
        [38].6   // LEVEL OVERFLOW main Tank
        [38].7   // ANORMAL EMPTY LEVEL main Tank
        [38].8   // temperature sensor default
        [38].9   // DEFAULT LOW LOW temperature DECAP
        [38].10   // DEFAULT LOW temperature DECAP
        [38].11   // DEFAULT HIGH temperature
        [38].12   // DEFAULT HIGH HIGH temperature DECAP
        [38].13   // DEFAULT NaOH transfert FROM OP008
        [38].14   // DEFAULT NaOH transfert FROM OP008
        [38].15   // DEFAULT NaOH fill up
        [39].0   // defaut gaswasser
        [39].1   // DEFAUT SERVOVANNE OUVERTURE CHAUFFE DECAP
        [39].2   // DEFAUT DECAP
        [39].3   // DEFAUT DECAP
        [39].4   // DEFAUT DECAP
        [39].5   // DEFAUT DECAP
        [39].6   // DEFAUT DECAP
        [39].7   // DEFAUT DECAP
        [39].8   // DEFAUT DECAP
        [39].9   // DEFAUT DECAP
        [39].10   // DEFAUT DECAP
        [39].11   // DEFAUT DECAP
        [39].12   // DEFAUT DECAP
        [39].13   // protection alim servovanne chaud decapage
        [39].14   // protection alim servovanne FROID decapage
        [39].15   // defaut vanne eau decap
        [41].0   // NEUTRAL defaut level haut
        [41].1   // NEUTRAL defaut level debordement haut
        [41].2   // neutral niveau trop bas
        [41].3   // defaut neutral ledigen
        [41].4   // DEFAUT ELECTR PMP 2 RINCAGE NEUTRAL
        [41].5   // LEVEL TOO HIGH rinse Tank
        [41].6   // LEVEL OVERFLOW rinse Tank
        [41].7   // ANORMAL EMPTY LEVEL rinse Tank
        [41].8   // Default filling up rinse Tank
        [41].9   // rinse conductivity sensor default
        [41].10   // DEF neutral
        [44].0   // LEVEL TOO HIGH main Tank
        [44].1   // LEVEL OVERFLOW main Tank
        [44].2   // ANORMAL EMPTY LEVEL main Tank
        [44].3   // temperature sensor default
        [44].4   // DEFAULT LOW LOW temperature ANO
        [44].5   // DEFAULT LOW temperature
        [44].6   // DEFAULT HIGH temperature
        [44].7   // DEFAULT HIGH HIGH temperature
        [44].8   // DEF ANOdisation
        [44].9   // DEF ANOdisation
        [44].10   // DEF ANOdisation
        [47].0   // temperature sensor default
        [47].1   // DEFAUT pompe 2 colo electrolyt
        [47].2   // DEFAUT mixer produit en prepa colo
        [47].3   // DEFAUT colo
        [47].4   // temperature OUT sensor default
        [47].5   // DEFAULT LOW LOW temperature KLEUR
        [47].6   // DEFAULT LOW temperature KLEUR
        [47].8   // DEFAULT HIGH HIGH temperature
        [50].0   // DEFAUT pompe 1 colo chimique
        [50].1   // DEFAUT pompe 2 colo chimique
        [50].2   // DEFAUT ventilo colo chimique
        [53].0   // temperature sensor in default
        [53].1   // DEFAUT SENSOR temp colmatage mil
        [53].2   // DEFAULT SENSOR t° out colmatage
        [53].3   // DEFAULT LOW LOW temperature
        [53].4   // DEFAULT LOW temperatuRE
        [53].5   // DEFAULT HIGH temperature
        [53].6   // DEFAULT HIGH HIGH temperature
        [53].7   // t° colm ne bouge plus
        [53].8   // niveau colmatage bas
        [53].9   // niveau colmatage haut
        [53].10   // niveau colmatage ledigen
        [65].0   // temperature sensor default
        [65].1   // DEFAULT LOW LOW temperature
        [65].2   // DEFAULT LOW temperature
        [65].3   // DEFAULT HIGHT temperature
        [65].4   // DEFAULT HIGHT HIGHT temperature
        [65].5   // DEFAUT FERMETURE SERVOVANNE
        [65].6   // DEFAUT OUVERTURE SERVOVANNE
        [65].7   // protection alimentation servovanne froid degraissage
        [68].0   // PMP 1 DECAP ELETRICAL FAULT
        [68].1   // PMP 2 DECAP ELETRICAL FAULT
        [68].2   // DECAPAGE VA 1 valve position default
        [68].3   // VA2 POSITION DEFAULT
        [68].4   // Fresh NaOH valve position default
        [68].5   // LEVEL OVERFLOW main Tank
        [68].6   // LEVEL OVERFLOW main Tank
        [68].7   // ANORMAL EMPTY LEVEL main Tank
        [68].8   // temperature sensor default
        [68].9   // DEFAULT LOW LOW temperature DECAP
        [68].10   // DEFAULT LOW temperature DECAP
        [68].11   // DEFAULT HIGH temperature
        [68].12   // DEFAULT HIGH HIGH temperature DECAP
        [68].13   // DEFAULT NaOH transfert FROM OP008
        [68].14   // DEFAULT NaOH transfert FROM OP008
        [68].15   // DEFAULT NaOH fill up
        [69].0   // DEFAUT SERVOVANNE CHAUFFE DECAP FERMETURE
        [69].1   // DEFAUT SERVOVANNE OUVERTURE CHAUFFE DECAP
        [69].2   // DEFAUT DECAP
        [69].3   // DEFAUT DECAP
        [69].4   // DEFAUT DECAP
        [69].5   // DEFAUT DECAP
        [69].6   // DEFAULT NaOH transfert to OP008
        [69].7   // DEFAUT DECAP
        [69].8   // DEFAUT DECAP
        [69].11   // DEFAUT DECAP
        [69].14   // DEFAUT DECAP
        [71].0   // NEUTRAL defaut level haut
        [71].1   // NEUTRAL defaut level debordement haut
        [71].2   // neutral niveau trop bas
        [71].3   // defaut neutral ledigen
        [71].4   // DEFAUT ELECTR PMP 2 RINCAGE NEUTRAL
        [71].5   // LEVEL TOO HIGH rinse Tank
        [71].6   // LEVEL OVERFLOW rinse Tank
        [71].7   // ANORMAL EMPTY LEVEL rinse Tank
        [71].8   // Default filling up rinse Tank
        [71].9   // rinse conductivity sensor default
        [71].10   // vanne apport eau RINCAGE NEUTRAL defaut
        [74].0   // LEVEL TOO HIGH main Tank
        [74].1   // LEVEL OVERFLOW main Tank
        [74].2   // ANORMAL EMPTY LEVEL main Tank
        [74].3   // temperature sensor default
        [74].4   // DEFAULT LOW LOW temperature ANO
        [74].5   // DEFAULT LOW temperature ANO
        [74].6   // DEFAULT HIGH temperature ANO
        [74].7   // DEFAULT HIGH HIGH temperature ANO
        [74].8   // DEFAUT ANO
        [74].9   // DEFAUT ANO
        [74].10   // DEFAUT ANO
        [77].0   // temperature sensor default
        [77].1   // DEFAUT pompe 2 colo electrolyt
        [77].2   // DEFAUT mixer produit en prepa colo
        [77].3   // DEFAUT COLO
        [77].4   // temperature OUT sensor default
        [77].5   // DEFAULT LOW LOW temperature KLEUR
        [77].6   // DEFAULT LOW temperature KLEUR
        [77].8   // DEFAULT HIGH HIGH temperature
        [80].0   // DEFAUT pompe 1 colo chimique
        [80].1   // DEFAUT pompe 2 colo chimique
        [80].2   // DEFAUT ventilo colo chimique
        [83].0   // temperature sensor in default
        [83].1   // DEFAUT SENSOR temp colmatage mil
        [83].2   // DEFAULT SENSOR t° out colmatage
        [83].3   // DEFAULT LOW LOW temperature colmat
        [83].4   // DEFAULT LOW temperatuRE
        [83].5   // DEFAULT HIGH temperature
        [83].6   // DEFAULT HIGH HIGH temperature
        [83].7   // t° colm ne bouge plus
        [83].8   // DEF COLM
        [83].9   // niveau colmatage haut
        [83].10   // niveau colmatage ledigen
   N200 : DINT[11];
   N21 : DINT[200] := ([66] := 310, [67] := 328, [68] := 373, [69] := 390, [70] := 420, [71] := 430, [72] := 470, [73] := 480, [74] := 345, [75] := 353, [76] := 382, [77] := 390, [82] := 910, [83] := 930, [84] := 970, [85] := 990);
        [66]   // SP TEMP LOW LOW temperature DEGRAIS
        [67]   // SP TEMP LOW temperature DEGRAIS
        [68]   // SP TEMP HIGH temperature DEGRAIS
        [69]   // SP TEMP HIGH HIGH temperature DEGRAIS
        [70]   // SP TEMP LOW LOW temperature DECAP
        [71]   // SP TEMP LOW temperature DECAP
        [72]   // SP TEMP HIGH temperature DECAP
        [73]   // SP TEMP HIGH HIGH temperature DECAP
        [74]   // SP TEMP LOW LOW temperature ANO
        [75]   // SP TEMP LOW temperature ANO
        [76]   // SP TEMP HIGH temperature ANO
        [77]   // SP TEMP HIGH HIGH temperature ANO
        [82]   // SP TEMP LOW LOW temperature COLAT
        [83]   // SP TEMP LOW temperature COLAT
        [84]   // SP TEMP HIGH temperature COLAT
        [85]   // SP TEMP HIGH HIGH temperature COLAT
   N7 : DINT[200] := ([3] := 32200, [6] := 1000, [8] := 940, [9] := 22, [10] := 50, [11] := 50, [12] := 50, [13] := 110, [14] := 5, [15] := 50, [16] := 1, [19] := 130, [20] := 50, [21] := -50, [22] := 35, [23] := -35, [26] := -32752, [28] := -48, [29] := 960, [30] := 965, [31] := 935, [33] := 22000, [40] := 5850, [45] := 200, [49] := 9558, [51] := 32200, [52] := 5850, [55] := 32767, [57] := 224, [58] := 5, [59] := 22, [60] := 1295, [61] := 40, [62] := 60, [63] := 20, [65] := 80, [66] := -80, [67] := 1000, [68] := 20, [70] := 45, [71] := -20, [72] := 2, [73] := 7, [74] := 137, [77] := 31, [78] := 1, [79] := 2, [80] := 824, [81] := 854, [82] := 850, [84] := 842, [87] := 450, [88] := 350, [90] := 2528, [94] := 429, [95] := 128, [96] := 145, [97] := 170, [98] := 990, [99] := 970,
        [100] := 500, [101] := 450, [102] := 970, [103] := 950, [105] := 985, [106] := 980, [107] := 990, [108] := 980, [109] := 995, [110] := 990, [111] := 995, [112] := 990, [121] := 1000, [123] := 370, [125] := 950, [126] := 120, [128] := 883, [154] := 886, [155] := 882, [160] := 680, [161] := 640, [162] := 940, [163] := 900, [164] := 740, [165] := 680, [166] := 980, [167] := 940, [170] := 500, [173] := 464, [178] := 375, [182] := 436, [184] := 204, [191] := 3, [192] := 3);
        [1]   // DEFAUT PRIORITE 1
        [2]   // defaut niveau 2
        [10]   // tour 1
        [10].0   // stock acide pas haut
        [10].1   // stock acide pas bas
        [10].2   // stock mazout pas haut
        [10].3   // stock mazout pas bas
        [10].4   // stock soude L1 pas haut
        [10].5   // stock soude L1 pas bas
        [10].7   // stock soude L2 pas bas
        [10].8   // stock soude L3 pas haut
        [10].9   // stock soude L3 pas bas
        [10].10   // PV vanne soude L1 fermée
        [10].13   // de PV chargement en cours
        [10].14   // DE PV BP EV SOUDE L1
        [11]   // tour 2
        [11].0   // DE PV BP EV SOUDE L3
        [11].1   // vers PV fuite stock mazout
        [11].2   // vers PV fuite stock acide
        [12]   // tour 3
        [13]   // consigne vitesse pour 3 ventilateurs
        [14]   // incrément vitesse pour ventilateurs
        [15]   // consigne vitesse par ventilateurs
        [16]   // Ecart T° tours refroidiss
        [17]   // position vanne decapage
        [19]   // T° précédente eau tour
        [20]   // Grand écart T° inc +
        [21]   // Grand écart T° inc -
        [22]   // petit écart T° inc +
        [23]   // petit écart T° inc -
        [25]   // quantité soude demandee
        [26].0   // vers plc stock demande de soude L3
        [26].1   // vers plc stock demande d'arret apport soude
        [26].2   // vers plc stock fc vanne apport soude décapage open
        [26].3   // vers plc stock apport soude finit
        [26].4   // vers plc stock fc vanne apport soudefermee
        [27]   // quantité acide demandee
        [28].0   // vers plc stock demande de acide
        [28].1   // vers plc stock demande d'arret apport acide
        [28].2   // vers plc stock fc vanne apport acide open
        [28].3   // vers plc stock apport acide finit
        [28].4   // vers plc stock fc vanne apport acid fermee
        [28].5   // fc vanne apport acide neutral open
        [28].6   // fc vanne apport acide neutral close
        [32]   // nombre de litre d'apport pour une quantite fixe d'adéox
        [33]   // limite low t°dec
        [34]   // limite high t°colm
        [35]   // limite low t°colm
        [36]   // limite h high t°dec
        [37]   // limite L low t°dec
        [38]   // limite H high t°ano
        [39]   // limite L low t°ano
        [40]   // limite H high t°colm
        [41]   // limite L low t°colm
        [42]   // aux temp colo
        [43]   // memo consigne coloration
        [45]   // de plc stock soude restante
        [46].3   // de plc stock ouverture vanne soude
        [46].4   // de plc stock apport soude finit
        [46].5   // de plc stock apport soude occupé
        [46].6   // de plc stock apport soude accordé
        [46].7   // de plc stock soude vers l1
        [46].8   // de plc stock soude vers L2
        [46].9   // de plc stock soude vers L3
        [46].10   // de plc stock soude vers L4
        [46].11   // de plc stock soude vers STAT
        [46].12   // DEFAULT NaOH fill up
        [47].3   // ouvrir vanne acide
        [47].4   // apport acide finit
        [47].5   // apport acide occupé
        [47].6   // apport acide accordé
        [47].7   // acide vers l1
        [47].8   // acide vers l2
        [47].9   // acide vers l3
        [47].10   // acide vers l4
        [47].11   // acide vers neut L1
        [47].12   // acide vers neut L2
        [47].13   // acide vers neut L3
        [47].14   // acide vers neut L4
        [48]   // quantite acide passé
        [49]   // consigne vanne refro
        [50]   // CONSIGNE MANU VANNE DEGRAISSAGE
        [51]   // CONSIGNE VANNE DEGRAISSAGE
        [52]   // consigne vanne chauffe decapage
        [53]   // consigne manuel vanne chauffe decapage
        [54]   // consigne manuel anne anoddisaton
        [55]   // consigne anne anoddisaton
        [60]   // poisit vanne DEGRAISSAGE
        [68]   // position vanne décapage chauffe
        [81]   // aux temp colm out
        [82]   // aux temp colm milieu
        [87]   // MEMO SP TEMP DECAP
        [88]   // MEMO SP TEMP DEGR
        [113]   // DIFFERENCE DE LVL DEPUIS LA DERNIERE MINUTE
        [121]   // limite max speed ven
        [122]   // nbr ventilo tour on
        [123]   // MEMO sp T° ano
        [126]   // MEMO LVL AANO
        [127]   // delta lvl colm
        [128]   // memo lvl colm
        [138]   // NOMBRE DEFAUT DEGRAISSAGE
        [139]   // MEMO DEFAUT DEGRAISSAGE
        [140]   // NUMBER DEFAULT FOR DECAP
        [141]   // MEMO DEF DECAP
        [142]   // NOMBRE DEFAUT NEUTRAL
        [143]   // MEMO DEFAUT NEUTRAL
        [144]   // NOMBRE DEFAUT ANO
        [145]   // MEMO DEF ANO
        [146]   // NOMBRE DEFAUT KLEUR C
        [147]   // MEMO DEFAUT KLEUR C
        [148]   // NOMBRE DEFAUT KLEUR E
        [149]   // MEMO DEFAUT KLEUR E
        [150]   // NOMBRE DEFAUT COLMAT
        [151]   // MEMO DEFAUT COLMAT
        [152]   // defaut algemeen
        [153]   // MEMO DEFAUT GENERAL
        [173]   // MEMO LVL DEC
        [174]   // DIFFERENCE DE LVL DEPUIS LA DERNIERE MINUTE
   N9 : DINT[200] := ([1] := 2881, [2] := 9873, [4] := 2, [8] := 30, [9] := 16353, [10] := 453, [11] := 842, [12] := 185, [13] := 346, [14] := 209, [15] := -2350, [16] := 1, [19] := 350, [20] := 450, [21] := 370, [22] := 1410, [23] := -63360, [24] := 950, [25] := 120, [26] := 1024, [29] := 210, [30] := 824, [31] := 854, [32] := 850, [33] := 20, [36] := 1, [38] := 1, [44] := 487, [45] := 250, [46] := 1648, [48] := 464, [49] := 302, [50] := 4096, [51] := 3650, [52] := 3700, [55] := 1000, [56] := 133, [57] := 1177, [58] := 975, [59] := 1, [60] := 447, [61] := 453, [64] := 50, [65] := 453, [66] := 435, [68] := 800, [69] := 883, [70] := 494, [71] := 422, [73] := 6, [76] := 10, [80] := 8192, [81] := 30, [82] := 9, [83] := 9, [84] := 137, [85] := 30, [88] := 7, [94] := 66, [95] := 350,
        [100] := 189, [101] := 210, [102] := 497, [103] := 361, [104] := 377, [105] := 366, [110] := 453);   // niveau decapage vers lancy (n9[10) ;;N9[70]
        [0]   // proceess VAriable PV
        [1]   // vers PV labo total eau tour
        [2]   // cond tour L3 vers PV labo
        [4]   // v bit
        [4].0   // /.
        [4].4   // DEFAULT NaOH transfert FROM OP008
        [4].5   // DEFAULT NaOH transfert FROM OP008
        [8].0   // de superv selection neutral
        [9]   // v bit
        [9].0   // VERS SUPERVIS CELLULE SORTIE
        [9].1   // DE superv L3 start soude
        [9].2   // DE superv L3 stop soude
        [9].3   // start acide
        [9].4   // stop acide
        [9].5   // on soude L1
        [9].6   // on soude L2
        [9].7   // on soude L3
        [9].8   // on soude L4
        [9].9   // on soude station
        [9].10   // on acide L1
        [9].11   // on acide L2
        [9].12   // on acide L3
        [9].13   // on acide L4
        [9].15   // new coil ftv
        [10]   // memo T°decapage
        [11]   // T° COLMATAGE
        [12]   // T° ANDISATION
        [13]   // T° DEgraissage
        [14]   // T°colo
        [15]   // TRACTION BS3
        [16]   // VITESSE
        [17]   // U REDRESSEUR 1
        [18]   // I REDRESSEUR 1
        [19]   // sp T° deg
        [20]   // sp t°dec
        [20].2   // change PV-SP to Sp-PV
        [21]   // sp T° ano
        [22]   // v bit
        [22].0   // DE PV MANU T° DEGRAISSAGE
        [22].1   // VERS PV OPEN VANNE T° DEGRAISSAGE
        [22].2   // VERS PV CLOSE VANNE T° DEGRAISSAGE
        [22].3   // DE PV MANU T° DECAPAGE
        [22].4   // VERS PV OPEN VANNE T° DECAPAGE
        [22].5   // VERS PV CLOSE VANNE T° DECAPAGE
        [22].6   // DE PV MANU T° ANODISATION
        [22].7   // VERS PV OPEN VANNE T° ANODISATION
        [22].8   // VERS PV CLOSE VANNE T° ANODISATION
        [22].9   // DE PV MANU T° COLMATAGE
        [22].10   // VERS PV OPEN VANNE T° COLMATAGE
        [22].11   // VERS PV CLOSE VANNE T° COLMATAGE
        [22].12   // DE PV OPEN VANNE T° DEGRAISSAGE
        [22].13   // DE PV CLOSE VANNE T° DEGRAISSAGE
        [22].14   // DE PV OPEN VANNE T° DECAPAGE
        [22].15   // DE PV CLOSE VANNE T° DECAPAGE
        [23]   // voir bits
        [23].0   // DE PV OPEN VANNE T° ANODISATION
        [23].1   // DE PV CLOSE VANNE T° ANODISATION
        [23].2   // DE PV OPEN VANNE T° COLMATAGE
        [23].3   // DE PV CLOSE VANNE T° COLMATAGE
        [23].4   // defaut level high ano
        [23].5   // defaut level low ano
        [23].6   // DE PV MANU T° colo
        [23].7   // DE PV OPEN VANNE T° colo
        [23].8   // DE PV CLOSE VANNE T° colo
        [23].9   // start stopt apport s
        [23].11   // fc vanne ano open
        [23].12   // fc vanne ano closed
        [23].13   // tour 1 on
        [23].14   // tour 2 on
        [23].15   // tour 3 on
        [24]   // sp t° colm
        [24].0   // sp t° colm
        [24].2   // sp t° colm
        [25]   // level ano
        [26]   // TRACTION
        [27]   // set point colo
        [28]   // position vanne coloration
        [29]   // total soude
        [30]   // t° in colmatage
        [31]   // t° out colmatage
        [32]   // temp colmatage milieu
        [33]   // position vanne décapage
        [34]   // U COLO
        [35]   // I COLO
        [36]   // U REDRESSEUR 2
        [37]   // I REDRESSEUR 2
        [38]   // U REDRESSEUR 3
        [39]   // I REDRESSEUR 3
        [40]   // U REDRESSEUR 4
        [41]   // I REDRESSEUR 4
        [42]   // DE superv L3 quantité soude
        [43]   // quantite soude pass
        [44]   // debit echangeur decapage soude
        [45]   // temp eau refroid
        [46]   // conduct tour
        [47]   // debit instantanné tour
        [48]   // level decapage
        [49]   // level neutral
        [50]   // high conduct
        [50].0   // vers superv niveau groupe hydraulique entrée
        [50].1   // vers superv niveau groupe hydraulique sortie
        [50].2   // defaut temperature total anodisation
        [50].3   // defaut temperature total decapage ligne 1,2,3
        [50].4   // TRS RAL
        [50].5   // VCN CXCBC
        [51]   // low conduct
        [52]   // high conduct
        [53]   // u colo
        [54]   // position vanne ano
        [55]   // position vanne colmatage 1
        [56]   // position vanne refroid decapage
        [57]   // POSITION VANNE DEGRAISSAGE
        [58]   // position vanne colmatage 2
        [59]   // I colo
        [61]   // csg vanne ano
        [62]   // csg vanne colm
        [63]   // i total redresseur
        [64]   // csg total vitesse ventilo
        [65]   // csg vanne chaudec
        [66]   // csg vanne froid dec
        [67]   // quantite acide demandé
        [68]   // quantite acide passé
        [69]   // level colmatage
        [71]   // vers lancy bits
        [72]   // VERS LANCY TOTALNaOH PASSER
        [73]   // VERS LANCY TOTALWATER PASSER
        [74]   // defaut niv 1
        [75]   // defaut niv 2
        [80]   // communication lancy
        [95]   // vers relalarm sp T° deg
        [100]   // total heure anodisation
        [101]   // total heure run lijn
        [102]   // total stop lijn
        [103]   // total heure anodisation
        [104]   // total heure run lijn
        [105]   // total stop lijn
   NCOM : INT[20] := ([0] := 464, [1] := 430, [3] := 4, [6] := 10, [11] := 2);
        [0]   // LVL DECAPAGE
        [1].0   // fc open vanne ano
        [11].6   // de lancy niv reactor too high
   new_def_decap : BOOL;
   offsetano : DINT := 2;
   offsetano_tdesc : DINT := 5;
   offsetano_Tup : DINT := 3;
   offsetdecfrois : DINT := 5;
   offstet_wkk : DINT := 40;
   ok_arm_io_decap : BOOL := 1;
   ok_dec_chauffe : BOOL;
   ok_dec_refroidir : BOOL;
   okpmpeau1 : BOOL := 1;
   okpmpeau2 : BOOL;
   okventilotour1 : BOOL := 1;
   okventilotour2 : BOOL := 1;
   okventilotour3 : BOOL := 1;
   ons1 : BOOL;
   ons2 : BOOL;
   ons3 : BOOL;
   ons4 : BOOL;
   ons5 : BOOL;
   ons6 : BOOL;
   ons7 : BOOL;
   ons8 : BOOL;
   ons9 : BOOL;
   out_v_ch_dec : REAL := 31208.0;
   par_p1_ano : DINT := 5;
   par_p2_ano : DINT := 10;
   par_p3_ano : DINT := 15;
   par_p4_ano : DINT := 20;
   par_p5_ano : DINT := 25;
   par_p6_ano : DINT := 30;
   par_rate_en_sec : DINT := 600;
   passage_jour_mois : BOOL;
   pid_ANO : PID := (CTL := -2113887104, EN := 1, CA := 1, INI := 1, OLL := 1, DVNA := 1, PVHA := 1, SP := 367.0, KP := 55.0, KI := 0.1, MAXS := 1000.0, DB := 0.01, MAXO := 100.0, UPD := 0.1, PV := 185.0, ERR := -182.0, MAXI := 1000.0, MAXCV := 1000.0, MAXTIE := 1000.0, DATA[0] := 44.00711, DATA[1] := 296.0, DATA[2] := 185.0, DATA[3] := -182.0, DATA[4] := 367.0, DATA[5] := 0.1, DATA[6] := 1.0, DATA[7] := 1.6, DATA[8] := 55.0, DATA[9] := 0.1, DATA[11] := 55.0, DATA[12] := 0.1, DATA[15] := 10.0, DATA[16] := 0.1);
   pid_colmat : PID := (CTL := -2147446144, EN := 1, INI := 1, OLH := 1, DVPA := 1, PVHA := 1, SP := 948.0, KP := 3.0, KI := 0.4, MAXS := 1000.0, DB := 1.0, SO := 100.0, MAXO := 100.0, UPD := 0.1, PV := 842.0, ERR := 106.0, OUT := 100.0, MAXI := 1000.0, MAXCV := 100.0, MAXTIE := 100.0, DATA[0] := 67.89783, DATA[1] := -1347.2001, DATA[2] := 842.0, DATA[3] := 106.0, DATA[4] := 948.0, DATA[5] := 0.1, DATA[6] := 1.0, DATA[7] := 1.6, DATA[8] := 3.0, DATA[9] := 0.4, DATA[11] := 3.0, DATA[12] := 0.4, DATA[15] := 1.0, DATA[16] := 1.0);
   pid_dec_ch : PID := (CTL := -2130672512, EN := 1, MO := 1, INI := 1, DVNA := 1, PVHA := 1, SP := 450.0, KP := 7.0, KI := 0.02, MAXS := 1000.0, DB := 3.0, MAXO := 100.0, UPD := 1.0, PV := 454.0, ERR := -4.0, MAXI := 1000.0, MAXCV := 100.0, MAXTIE := 4095.0, DATA[0] := 2.8, DATA[1] := -726.4, DATA[2] := 454.0, DATA[3] := -4.0, DATA[4] := 450.0, DATA[5] := 0.1, DATA[6] := 1.0, DATA[7] := 16.0, DATA[8] := 7.0, DATA[9] := 0.02, DATA[11] := 7.0, DATA[12] := 0.02, DATA[15] := 1.0, DATA[16] := 0.024420025);
   pid_dec_fr : PID := (CTL := -2113893248, EN := 1, CA := 1, INI := 1, EWD := 1, DVNA := 1, PVHA := 1, SP := 455.0, KP := 17.0, KI := 0.014, BIAS := 10.0, MAXS := 1000.0, DB := 2.0, SO := 13.944649, MAXO := 100.0, MINO := 6.0, UPD := 1.0, PV := 454.0, ERR := -1.0, OUT := 13.944649, MAXI := 1000.0, MAXCV := 1000.0, MAXTIE := 4095.0, DATA[0] := 3.9446487, DATA[1] := 726.4, DATA[2] := 454.0, DATA[3] := -1.0, DATA[4] := 455.0, DATA[5] := 0.1, DATA[6] := 1.0, DATA[7] := 16.0, DATA[8] := 17.0, DATA[9] := 0.014, DATA[11] := 17.0, DATA[12] := 0.014, DATA[15] := 10.0, DATA[16] := 0.024420025);
   pid_deg : PID := (CTL := -2147446144, EN := 1, INI := 1, OLH := 1, DVPA := 1, PVHA := 1, SP := 350.0, KP := 7.5, KI := 420.0, MAXS := 1000.0, DB := 2.0, SO := 100.0, MAXO := 100.0, UPD := 0.1, PV := 346.0, ERR := 4.0, OUT := 100.0, MAXI := 1000.0, MAXCV := 100.0, MAXTIE := 100.0, DATA[0] := 96.470184, DATA[1] := -553.60004, DATA[2] := 346.0, DATA[3] := 4.0, DATA[4] := 350.0, DATA[5] := 0.1, DATA[6] := 1.0, DATA[7] := 1.6, DATA[8] := 7.5, DATA[9] := 420.0, DATA[11] := 7.5, DATA[12] := 420.0, DATA[15] := 1.0, DATA[16] := 1.0);
   pid_pmpANO : PID := (CTL := -2097118080, EN := 1, CA := 1, MO := 1, INI := 1, DVNA := 1, PVHA := 1, SP := 370.0, KP := 25.0, KI := 0.08, MAXS := 1000.0, DB := 2.0, MAXO := 100.0, UPD := 0.1, PV := 185.0, ERR := -185.0, MAXI := 1000.0, MAXCV := 1000.0, MAXTIE := 1000.0, DATA[0] := 462.5, DATA[1] := 296.0, DATA[2] := 185.0, DATA[3] := -185.0, DATA[4] := 370.0, DATA[5] := 0.1, DATA[6] := 1.0, DATA[7] := 1.6, DATA[8] := 25.0, DATA[9] := 0.08, DATA[11] := 25.0, DATA[12] := 0.08, DATA[15] := 10.0, DATA[16] := 0.1);
   pid_pmprenvoi : PID := (CTL := -2147449984, EN := 1, INI := 1, DVPA := 1, PVLA := 1, PVHA := 1, SP := 90.0, KP := 40.0, KI := 0.8, MAXS := 1000.0, DB := 5.0, SO := 100.0, MAXO := 100.0, UPD := 0.1, ERR := 90.0, OUT := 100.0, MAXI := 1000.0, MAXCV := 1000.0, MAXTIE := 4095.0, DATA[0] := -260.0, DATA[3] := 90.0, DATA[4] := 90.0, DATA[5] := 0.1, DATA[6] := 1.0, DATA[7] := 1.6, DATA[8] := 40.0, DATA[9] := 0.8, DATA[11] := 40.0, DATA[12] := 0.8, DATA[15] := 10.0, DATA[16] := 0.024420025);
   PIDwkk : PID := (CTL := -2147446144, EN := 1, INI := 1, OLH := 1, DVPA := 1, PVHA := 1, SP := 950.0, KP := 300.0, KI := 0.01, MAXS := 1000.0, SO := 100.0, MAXO := 100.0, MINO := 99.0, UPD := 0.1, PV := 842.0, ERR := 108.0, OUT := 100.0, MAXI := 1000.0, MAXCV := 100.0, MAXTIE := 4095.0, DATA[0] := 69.99999, DATA[1] := -1347.2001, DATA[2] := 842.0, DATA[3] := 108.0, DATA[4] := 950.0, DATA[5] := 0.1, DATA[6] := 1.0, DATA[7] := 1.6, DATA[8] := 300.0, DATA[9] := 0.01, DATA[11] := 300.0, DATA[12] := 0.01, DATA[15] := 1.0, DATA[16] := 0.024420025);
   pmp_vid_colmat : BOOL := 1;
   pmpano_inhold : BOOL;
   pmpano_inholdval : DINT := 325;
   pmprenv_inhold : BOOL := 1;
   pmprenv_inholdval : DINT := 1000;
   POS_V_COLO : DINT;
   POS_V_DEC : DINT := 20;
   pour_offset_wkk : REAL := 1.0;
   PV_PID_COLM : DINT;
   R6 : CONTROL[10];
   refroidis_fort : BOOL;
   regul_anob : BOOL := 1;
   S : INT[164] := ([0] := 16#0004, [1] := 16#00b6, [2] := 16#1012, [3] := 16#a003, [4] := 16#cf5d, [5] := 16#4000, [6] := 16#0021, [11] := 16#ffff, [12] := 16#ffff, [14] := 16#010e, [15] := 16#0b18, [17] := 16#0002, [20] := 16#0008, [21] := 16#0003, [22] := 16#0005, [23] := 16#0003, [27] := 16#ffff, [28] := 16#ffff, [30] := 16#000a, [31] := 16#000b, [33] := 16#0288, [34] := 16#0002, [35] := 16#001a, [37] := 16#07e1, [38] := 16#0001, [39] := 16#001e, [40] := 16#000a, [41] := 16#0012, [42] := 16#0020, [43] := 16#e091, [53] := 16#0003, [57] := 16#0191, [58] := 16#0002, [59] := 16#0004, [60] := 16#021d, [61] := 16#0002, [62] := 16#0007, [63] := 16#0401, [64] := 16#0023, [65] := 16#0010, [66] := 16#0200, [83] := 16#0046, [84] := 16#f901, [85] := 16#0001, [86] := 16#01a3);
   S_bP_dmd_man_pmp_eau : BOOL;
   S_BP_manu_DEC : BOOL;
   s_bp_neutral : BOOL;
   s_bp_stop_acide : BOOL;
   s_bp_stop_soude : BOOL;
   s_bp_strt_acide : BOOL;
   s_bp_strt_soude : BOOL;
   S_C_TOUR : DINT := 1648;
   S_COND_TOUR : DINT := 1648;
   S_csg_manu_dec_ch : DINT := 100;
   S_csg_manu_Dec_froid : DINT;
   S_csg_manu_Dec_froid1 : REAL;
   S_CSG_SPD_PMP_WKK : DINT := 1000;
   s_csg_ventilo_ano : DINT;
   s_def_new : DINT;
   s_def_old : DINT;
   S_def_pmp_decap_1 : BOOL := 1;
   S_def_pmp_decap_2 : BOOL := 1;
   S_def_pmpeauano1 : BOOL := 1;
   S_def_pmpeauano2 : BOOL;
   S_def_ventilo_eau1 : BOOL := 1;
   S_def_ventilo_eau2 : BOOL := 1;
   S_def_ventilo_eau3 : BOOL := 1;
   S_FLOW_RETURN_LANCY : DINT := 90;
   S_FLOW_TOUR : DINT;
   S_FLW_ech_DECAP : DINT := 487;
   S_FLW_XCHG_DECAP : DINT := 487;
   S_hiver : BOOL := 1;
   S_I_COL : DINT;
   S_I_COLO : DINT;
   S_I_R1 : DINT;
   S_I_R2 : DINT;
   S_I_R3 : DINT;
   S_I_R4 : DINT;
   S_IR1 : DINT;
   S_LVL_ANO : DINT := 120;
   S_LVL_COLMAT : DINT := 883;
   S_LVL_DECAP : DINT := 464;
   S_LVL_NEUT : DINT := 302;
   S_MA_PMP_WKK : BOOL := 1;
   S_MAN_PMP_WKK : BOOL := 1;
   s_nbr_ventilo_ano : DINT;
   S_niv_ANO : DINT := 120;
   s_pos_dec_ch : REAL := 20.308594;
   S_pos_dec_FR : REAL := 132.78326;
   S_Q_DEM_h2so4 : DINT;
   S_Q_DEM_NAOH : DINT;
   S_Q_PAS_NAOH : DINT;
   S_q_pass_h2so4 : DINT := 800;
   S_RUN_PMP_DEC1 : BOOL := 1;
   S_RUN_PMP_DEC2 : BOOL := 1;
   S_run_pmpeauano1 : BOOL := 1;
   S_run_pmpeauano2 : BOOL;
   S_run_ventilo_1 : BOOL;
   s_run_ventilo_2 : BOOL;
   S_run_ventilo_3 : BOOL;
   S_SP_ANO : DINT := 370;
   S_SP_COLO : DINT;
   S_SP_DEC : DINT := 450;
   S_SP_DEGRAIS : DINT := 350;
   S_SP_T_COLMAT : DINT := 950;
   S_SPD_PMP_WKK : DINT;
   S_SPEED : DINT := 1;
   s_T_2_DEC : REAL := 453.3235;
   S_T_ANO : DINT := 185;
   S_T_AVER_COLM : DINT := 842;
   S_T_COLO : DINT := 210;
   S_T_DEC : DINT := 1000;
   S_T_DEC2 : DINT := 454;
   S_T_DEC3 : REAL := 454.56738;
   S_T_DEGRAIS : DINT := 346;
   S_T_EAU_REFROID : DINT := 250;
   S_T_ent_COLM : DINT := 824;
   S_T_IN_COLMAT : DINT := 824;
   S_T_MID_COLMAT : DINT := 850;
   S_T_moy_COLM : DINT := 842;
   S_T_OUT_COLMAT : DINT := 854;
   S_TEMPS_ANODIS : DINT := 189;
   S_TEMPS_RUN_LINE : DINT := 210;
   S_TEMPS_RUN_LINE_LAST_MONTH : DINT := 377;
   S_TEMPS_STOP_LINE : DINT := 497;
   S_TEMPS_STOP_LINE_LAST_MONTH : DINT := 366;
   S_TOT_I : DINT;
   S_TPS_ANO_LAST_MONTH : DINT := 361;
   S_TRACT : DINT := 1024;
   S_TRACT_BS3 : DINT := -2350;
   S_U_COLO : DINT;
   S_U_R1 : DINT;
   S_U_R2 : DINT := 1;
   S_U_R3 : DINT := 1;
   S_U_R4 : DINT;
   scp_cond_tour : SCP := (Input := 4340.0, Input_Min := 3277.0, Input_Max := 16384.0, Scaled_Min := 10.0, Scaled_Max := 20000.0, Output := 1631.223);
   SCP_CV_ANO : SCP := (Input_Max := 1000.0, Scaled_Max := 200.0);
   scp_CV_ch_dec : SCP := (Input := 31000.0, Input_Max := 31000.0, Scaled_Min := 1000.0);
   SCP_CV_COLMAT : SCP := (Input := 100.0, Input_Max := 100.0, Scaled_Max := 32767.0, Output := 32767.002);
   SCP_CV_DEC_CH : SCP := (Input_Max := 100.0, Scaled_Min := 31208.0, Scaled_Max := 6242.0, Output := 31208.0);
   SCP_CV_DEG : SCP := (Input := 100.0, Input_Max := 100.0, Scaled_Max := 32200.0, Output := 32200.0);
   SCP_CV_VENTILO : SCP := (Input := 50.0, Input_Max := 1000.0, Scaled_Max := 1000.0, Output := 50.0);
   scp_CV_wkk : SCP := (Input := 3277.0, Input_Min := 3277.0, Input_Max := 16384.0, Scaled_Max := 1000.0);
   SCP_FLW_TOUR : SCP := (Input := 3277.0, Input_Min := 3277.0, Input_Max := 16384.0, Scaled_Max := 100.0);
   scp_I_colo : SCP := (Input := 3286.0, Input_Min := 3277.0, Input_Max := 16383.0, Scaled_Max := 1000.0, Output := 0.6867084);
   scp_I_r1 : SCP := (Input := 3277.0, Input_Min := 3277.0, Input_Max := 16383.0, Scaled_Max := 170.0);
   scp_I_r2 : SCP := (Input := 3278.0, Input_Min := 3277.0, Input_Max := 16383.0, Scaled_Max := 170.0, Output := 0.012971158);
   scp_I_r3 : SCP := (Input := 3277.0, Input_Min := 3277.0, Input_Max := 16383.0, Scaled_Max := 170.0);
   SCP_I_R4 : SCP := (Input := 3276.0, Input_Min := 3277.0, Input_Max := 16383.0, Scaled_Max := 170.0, Output := -0.012971158);
   SCP_LVL_ANO : SCP := (Input := 4849.0, Input_Min := 3277.0, Input_Max := 16384.0, Scaled_Max := 1000.0, Output := 119.935905);
   SCP_LVL_COLM : SCP := (Input := 14862.0, Input_Min := 3277.0, Input_Max := 16384.0, Scaled_Max := 1000.0, Output := 883.87885);
   SCP_LVL_DEC : SCP := (Input := 4134.0, Input_Min := 3277.0, Input_Max := 16384.0, Scaled_Max := 1000.0, Output := 65.38491);
   scp_out_v_ch_dec : SCP := (Input := 5850.0, Input_Min := 5850.0, Input_Max := 31850.0, Scaled_Min := 31208.0, Scaled_Max := 6242.0, Output := 31208.0);
   scp_pmp_decap_1 : SCP := (Input := 300.0, Input_Max := 1000.0, Scaled_Max := 10500.0, Output := 3150.0);
   scp_pmp_decap_2 : SCP := (Input := 1000.0, Input_Max := 1000.0, Scaled_Max := 10500.0, Output := 10500.0);
   scp_pos_v_ch_dec : SCP := (Input := 16130.0, Input_Min := 3680.0, Input_Max := 16384.0, Scaled_Min := 1000.0, Output := 19.993774);
   scp_pos_Vroid_dec : SCP := (Input := 5035.0, Input_Min := 3295.0, Input_Max := 16384.0, Scaled_Max := 1000.0, Output := 132.93607);
   scp_t_2_dec : SCP := (Input := 14739.0, Input_Max := 32511.0, Scaled_Max := 1000.0, Output := 453.35425);
   SCP_T_ANO : SCP := (Input := 5699.0, Input_Min := 3277.0, Input_Max := 16383.0, Scaled_Max := 1000.0, Output := 184.80086);
   SCP_T_DEC : SCP := (Input := 16384.0, Input_Min := 3277.0, Input_Max := 16383.0, Scaled_Max := 1000.0, Output := 1000.07635);
   scp_T_deg : SCP := (Input := 7981.0, Input_Min := 3277.0, Input_Max := 16383.0, Scaled_Max := 1000.0, Output := 358.9196);
   SCP_T_EAU_REFR : SCP := (Input_Min := 3277.0, Input_Max := 16384.0, Scaled_Max := 1000.0, Output := -250.01907);
   SCP_T_IN_COLM : SCP := (Input := 14080.0, Input_Min := 3277.0, Input_Max := 16384.0, Scaled_Max := 1000.0, Output := 824.21606);
   SCP_T_MIL_COLM : SCP := (Input := 14341.0, Input_Min := 3277.0, Input_Max := 16384.0, Scaled_Max := 1000.0, Output := 844.1291);
   SCP_T_OUT_COLM : SCP := (Input := 14470.0, Input_Min := 3277.0, Input_Max := 16384.0, Scaled_Max := 1000.0, Output := 853.9711);
   SCP_TRACT : SCP := (Input_Min := 3277.0, Input_Max := 16383.0, Scaled_Max := 9400.0, Output := -2350.3586);
   scp_u_colo : SCP := (Input := 3277.0, Input_Min := 3277.0, Input_Max := 16383.0, Scaled_Max := 1000.0);
   scp_u_r1 : SCP := (Input := 3285.0, Input_Min := 3277.0, Input_Max := 16383.0, Scaled_Max := 500.0, Output := 0.30520374);
   scp_u_r2 : SCP := (Input := 3295.0, Input_Min := 3277.0, Input_Max := 16383.0, Scaled_Max := 500.0, Output := 0.6867084);
   scp_u_r3 : SCP := (Input := 3307.0, Input_Min := 3277.0, Input_Max := 16383.0, Scaled_Max := 500.0, Output := 1.144514);
   SCP_U_R4 : SCP := (Input := 3277.0, Input_Min := 3277.0, Input_Max := 16383.0, Scaled_Max := 500.0);
   scp_Vanne_manu : SCP;
   scp_Vanne_Vroid_dec : SCP := (Input := 139.0, Input_Max := 1000.0, Scaled_Min := 6500.0, Scaled_Max := 28500.0, Output := 9558.0);
   scp_ventilo : SCP := (Input_Max := 1000.0, Scaled_Min := 6242.0, Scaled_Max := 25000.0, Output := 6242.0);
   stat_L3 : DINT[20] := ([1] := 589824, [3] := 800, [4] := 2, [5] := 757);
        [0]   // de plc stock soude restante
        [1].3   // de plc stock ouverture vanne soude
        [1].4   // de plc stock apport soude finit
        [1].5   // de plc stock apport soude occupé
        [1].6   // de plc stock apport soude accordé
        [1].7   // de plc stock soude vers l1
        [1].8   // de plc stock soude vers L2
        [1].9   // de plc stock soude vers L3
        [1].10   // de plc stock soude vers L4
        [1].11   // de plc stock soude vers STAT
        [1].12   // DEFAULT NaOH fill up
        [2].3   // ouvrir vanne acide
        [2].4   // apport acide finit
        [2].5   // apport acide occupé
        [2].6   // apport acide accordé
        [2].7   // acide vers l1
        [2].8   // acide vers l2
        [2].9   // acide vers l3
        [2].10   // acide vers l4
        [2].11   // acide vers neut L1
        [2].12   // acide vers neut L2
        [2].13   // acide vers neut L3
        [2].14   // acide vers neut L4
        [2].15   // quantite acide passé
   Status : INT := 12640;   // INT tag to retrieve Status value through GSV created during conversion
   T4 : TIMER[180] := ([1].PRE := 800, [2].PRE := 800, [3].PRE := 20000, [4].PRE := 20000, [4].ACC := 20000, [4].EN := 1, [4].DN := 1, [5].PRE := 4000, [5].ACC := 4000, [5].EN := 1, [5].DN := 1, [6].PRE := 450, [6].ACC := 500, [7].PRE := 10000, [8].PRE := 1500, [9].PRE := 3000, [10].PRE := 3000, [11].PRE := 3000, [12].PRE := 1000, [13].PRE := 600, [13].ACC := 600, [14].PRE := 3000, [15].PRE := 20000, [16].PRE := 20000, [16].ACC := 20000, [16].EN := 1, [16].DN := 1, [17].PRE := 1500, [18].PRE := 5000, [19].PRE := 6000, [20].PRE := 6000, [21].PRE := 4000, [22].PRE := 50, [22].ACC := 100, [23].PRE := 600, [23].ACC := 600, [24].PRE := 20000, [25].PRE := 70000, [25].ACC := 70000, [25].EN := 1, [25].DN := 1, [26].PRE := 10000, [27].PRE := 150, [27].ACC := 200, [28].PRE := 5000, [29].PRE := 120000, [29].ACC := 120000, [30].PRE := 360000, [30].ACC := 360000, [31].PRE := 3600000, [31].ACC := 65500, [31].EN := 1, [31].TT := 1, [32].PRE := 600000, [32].ACC := 600000, [33].PRE := 5000, [33].ACC := 1600, [33].EN := 1, [33].TT := 1, [34].PRE := 1800000,
        [35].PRE := 60000, [35].ACC := 60000, [36].PRE := 60000, [37].PRE := 3600000, [37].ACC := 65500, [37].EN := 1, [37].TT := 1, [38].PRE := 30000, [38].ACC := 8000, [38].EN := 1, [38].TT := 1, [39].PRE := 180000, [39].ACC := 27000, [39].EN := 1, [39].TT := 1, [40].PRE := 60000, [40].ACC := 36401, [40].EN := 1, [40].TT := 1, [41].PRE := 60000, [41].EN := 1, [41].DN := 1, [42].PRE := 60000, [42].ACC := 29000, [42].EN := 1, [42].TT := 1, [43].PRE := 60000, [43].EN := 1, [43].DN := 1, [44].PRE := 60000, [44].EN := 1, [44].DN := 1, [45].PRE := 60000, [45].EN := 1, [45].DN := 1, [46].PRE := 1800000, [47].PRE := 5400000, [47].ACC := 5400000, [48].PRE := 1500000, [48].ACC := 1500000, [49].PRE := 3600000, [49].ACC := 36500, [49].EN := 1, [49].TT := 1, [50].PRE := 15000, [51].PRE := 15000, [52].PRE := 240000, [53].PRE := 4000, [53].ACC := 3600, [53].EN := 1, [53].TT := 1, [54].PRE := 700, [55].PRE := 1500, [55].ACC := 1000, [55].EN := 1, [55].DN := 1, [56].PRE := 500, [57].PRE := 5000, [58].PRE := 1500000, [58].ACC := 1500000,
        [59].PRE := 4000, [59].ACC := 4000, [59].EN := 1, [59].DN := 1, [62].PRE := 1200000, [63].PRE := 60000, [63].ACC := 60000, [64].PRE := 900000, [65].PRE := 1200000, [66].PRE := 900000, [67].PRE := 900000, [68].PRE := 1200000, [68].ACC := 1200000, [68].EN := 1, [68].DN := 1, [69].PRE := 1200000, [69].ACC := 1200000, [69].EN := 1, [69].DN := 1, [70].PRE := 1200000, [70].ACC := 1200000, [70].EN := 1, [70].DN := 1, [71].PRE := 1200000, [71].ACC := 1200000, [71].EN := 1, [71].DN := 1, [72].PRE := 240000, [73].PRE := 240000, [74].PRE := 240000, [75].PRE := 600000, [75].ACC := 600000, [76].PRE := 240000, [77].PRE := 240000, [78].PRE := 240000, [79].PRE := 120000, [80].PRE := 1200, [81].PRE := 120000, [82].PRE := 120000, [84].PRE := 120000, [85].PRE := 300000, [86].PRE := 300000, [88].PRE := 10000, [89].PRE := 10000, [90].PRE := 3600000, [90].ACC := 3540200, [91].PRE := 3600000, [91].ACC := 1566500, [92].PRE := 3600000, [92].ACC := 910200, [92].EN := 1, [92].TT := 1, [93].PRE := 30000, [93].ACC := 8000, [93].EN := 1, [93].TT := 1, [95].PRE := 150000, [95].ACC := 128800, [95].EN := 1, [95].TT := 1,
        [96].PRE := 60000, [96].ACC := 40300, [96].EN := 1, [96].TT := 1, [97].PRE := 30000, [97].ACC := 30000);
        [2]   // test
        [30].PRE   // mul par 28000 au départ 23/10/14 180000 le 14/9/2016 - > 234000
   T_DEC : DINT;
   T_EAU_REFROID : REAL := -250.01907;
   T_IN_COLMAT : DINT := 825;
   T_man_pmp_eau : TIMER := (PRE := 1800000, ACC := 65000, TT := 1, DN := 1);
   T_MIL_COLMAT : REAL := 843.7476;
   t_minute : TIMER := (PRE := 60000, ACC := 29100, EN := 1, TT := 1);   // tempo on toutes les minute
   T_OUT_COLMAT : REAL := 854.1237;
   T_pmp_decap_1 : TIMER := (PRE := 30000, ACC := 30000, EN := 1, DN := 1);
   T_pmp_decap_2 : TIMER := (PRE := 30000, ACC := 30000, EN := 1, DN := 1);
   T_pmpeau_1 : TIMER := (PRE := 10000, ACC := 10000, EN := 1, DN := 1);
   T_pmpeau_2 : TIMER := (PRE := 20000);
   t_seconde : TIMER := (PRE := 1000);   // tempo on toutes les secondes
   T_ventilo_eau_1 : TIMER := (PRE := 30000);
   T_ventilo_eau_2 : TIMER := (PRE := 30000);
   T_ventilo_eau_3 : TIMER := (PRE := 30000);
   tcligno : TIMER := (PRE := 1000);
   test : BOOL;
   test1 : REAL;
   test2 : REAL := 446.51813;
   test3 : REAL := 293022.34;
   test4 : DINT := 293;
   test5 : DINT := 1000;
   TIE_PID_wkk : DINT;
   TRACT : REAL := -2350.3586;
   U_R1 : REAL := 0.30520374;
   U_R2 : DINT := 1;
   U_R3 : DINT := 1;
   U_R4 : REAL := 0.076300934;
   vit_pmp_dec_1 : REAL := 300.0;
   vit_pmp_dec_2 : DINT := 1000;
   vit_renvoi_lancy : DINT := 300;
   vit_ventilo : DINT;
   vitpmpeau : DINT := 500;
   Vroid_dec : SCP;
   water_flow_from_ibt : REAL;
   wkk5 : REAL := 1.8310826;
   wkk_L3 : DINT[125] := ([3] := 5, [12] := 6565);
        [9].0   // run pmp de wkk
END_VAR
